REGION Network 36: LT-502 BUFF
   RUNG wire#powerrail
      Contact( "AlwaysTRUE" )
      wire#w1
      { S7_Templates := "SrcType := Real" } LT_Contact(in1 := "AI SCALING DB".PV."LEVEL TRANSMITTER 502", in2 := "AI SCALING DB"."LT-502 SET VALVE".LL)
      { S7_Templates := "time_type := Time" } "IEC_Timer_0_DB_30".TON(pt := T#3S, et =>)
      Move(in := 1, out1 => "AI SCALING DB"."LT-502".LOW_BUFF)
   END_RUNG
   RUNG wire#w1
      { S7_Templates := "SrcType := Real" } GE_Contact(in1 := "AI SCALING DB".PV."LEVEL TRANSMITTER 502", in2 := "AI SCALING DB"."LT-502 SET VALVE".L)
      { S7_Templates := "time_type := Time" } "IEC_Timer_0_DB_31".TON(pt := T#3S, et =>)
      Move(in := 2, out1 => "AI SCALING DB"."LT-502".LOW_BUFF)
   END_RUNG
   RUNG wire#w1
      { S7_Templates := "SrcType := Real" } LT_Contact(in1 := "AI SCALING DB".PV."LEVEL TRANSMITTER 502", in2 := "AI SCALING DB"."LT-502 SET VALVE".H)
      { S7_Templates := "time_type := Time" } "IEC_Timer_0_DB_32".TON(pt := T#3S, et =>)
      Move(in := 3, out1 => "AI SCALING DB"."LT-502".HIGH_BUFF)
   END_RUNG
   RUNG wire#w1
      { S7_Templates := "SrcType := Real" } GE_Contact(in1 := "AI SCALING DB".PV."LEVEL TRANSMITTER 502", in2 := "AI SCALING DB"."LT-502 SET VALVE".HH)
      { S7_Templates := "time_type := Time" } "IEC_Timer_0_DB_33".TON(pt := T#3S, et =>)
      Move(in := 4, out1 => "AI SCALING DB"."LT-502".HIGH_BUFF)
   END_RUNG
   // the same network as SCL:
   "IEC_Timer_0_DB_30".TON(IN := "AlwaysTRUE" AND ("AI SCALING DB".PV."LEVEL TRANSMITTER 502" < "AI SCALING DB"."LT-502 SET VALVE".LL),
                           PT := T#3S);
   IF "IEC_Timer_0_DB_30".Q THEN "AI SCALING DB"."LT-502".LOW_BUFF := 1; END_IF;
   "IEC_Timer_0_DB_31".TON(IN := "AlwaysTRUE" AND ("AI SCALING DB".PV."LEVEL TRANSMITTER 502" >= "AI SCALING DB"."LT-502 SET VALVE".L),
                           PT := T#3S);
   IF "IEC_Timer_0_DB_31".Q THEN "AI SCALING DB"."LT-502".LOW_BUFF := 2; END_IF;
   "IEC_Timer_0_DB_32".TON(IN := "AlwaysTRUE" AND ("AI SCALING DB".PV."LEVEL TRANSMITTER 502" < "AI SCALING DB"."LT-502 SET VALVE".H),
                           PT := T#3S);
   IF "IEC_Timer_0_DB_32".Q THEN "AI SCALING DB"."LT-502".HIGH_BUFF := 3; END_IF;
   "IEC_Timer_0_DB_33".TON(IN := "AlwaysTRUE" AND ("AI SCALING DB".PV."LEVEL TRANSMITTER 502" >= "AI SCALING DB"."LT-502 SET VALVE".HH),
                           PT := T#3S);
   IF "IEC_Timer_0_DB_33".Q THEN "AI SCALING DB"."LT-502".HIGH_BUFF := 4; END_IF;
END_REGION

REGION Network 38: "DataToSlave".DATA1."LT-502 BUFFER"."LT-502 LOW"
   RUNG wire#powerrail
      Move(in := "AI SCALING DB"."LT-502".LOW_BUFF, out1 => "DataToMaster".DATA1."LT-502".LOW_BUFF)
   END_RUNG
   // the same network as SCL:
   "DataToMaster".DATA1."LT-502".LOW_BUFF := "AI SCALING DB"."LT-502".LOW_BUFF;
END_REGION

REGION Network 39: "DataToSlave".DATA1."LT-502 BUFFER"."LT-502 HIGH
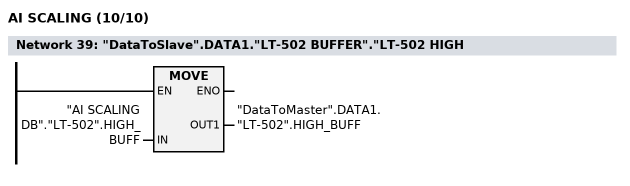
   RUNG wire#powerrail
      Move(in := "AI SCALING DB"."LT-502".HIGH_BUFF, out1 => "DataToMaster".DATA1."LT-502".HIGH_BUFF)
   END_RUNG
   // the same network as SCL:
   "DataToMaster".DATA1."LT-502".HIGH_BUFF := "AI SCALING DB"."LT-502".HIGH_BUFF;
END_REGION
END_FUNCTION

FUNCTION_BLOCK "SCALE"   // FB1, LAD
{ S7_Optimized_Access := 'TRUE' }
// stored: MemoryReserve 100, SetENOAutomatically false
   VAR_INPUT
      "SCALE MIN" : Real;
      "SCALE MAX" : Real;
      INPUT : Int;
      "RAW MIN" : Int;
      "RAW MAX" : Int;
   END_VAR
   VAR_OUTPUT
      "PV VALUE" : Real;
   END_VAR
   VAR_TEMP
      NORMX : Real;
   END_VAR
BEGIN

REGION Network 1
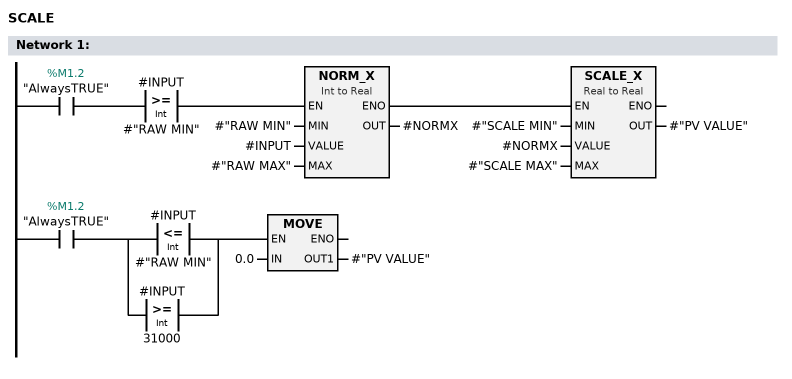
   RUNG wire#powerrail
      Contact( "AlwaysTRUE" )
      { S7_Templates := "SrcType := Int" } GE_Contact(in1 := #INPUT, in2 := #"RAW MIN")
      { S7_Templates := "[SrcType := Int, DestType := Real]" } Normalize(min := #"RAW MIN", value := #INPUT, max := #"RAW MAX", out => #NORMX)
      { S7_Templates := "[SrcType := Real, DestType := Real]" } Scale(min := #"SCALE MIN", value := #NORMX, max := #"SCALE MAX", out => #"PV VALUE")
   END_RUNG
   RUNG wire#powerrail
      Contact( "AlwaysTRUE" )
      wire#w1
      { S7_Templates := "SrcType := Int" } LE_Contact(in1 := #INPUT, in2 := #"RAW MIN")
      wire#w2
      Move(in := 0.0, out1 => #"PV VALUE")
   END_RUNG
   RUNG wire#w1
      { S7_Templates := "SrcType := Int" } GE_Contact(in1 := #INPUT, in2 := 31000)
   END_RUNG wire#w2
   // the same network as SCL:
   IF "AlwaysTRUE" AND (#INPUT >= #"RAW MIN") THEN
       #NORMX := NORM_X(MIN := #"RAW MIN", VALUE := #INPUT, MAX := #"RAW MAX");
       #"PV VALUE" := SCALE_X(MIN := #"SCALE MIN", VALUE := #NORMX, MAX := #"SCALE MAX");
   END_IF;
   IF "AlwaysTRUE" AND ((#INPUT <= #"RAW MIN") OR (#INPUT >= 31000)) THEN #"PV VALUE" := 0.0; END_IF;
END_REGION
END_FUNCTION_BLOCK

FUNCTION "INPUT MAPING" : Void   // FC1, LAD
{ S7_Optimized_Access := 'TRUE' }
// stored: SetENOAutomatically false
BEGIN

REGION Network 1: "CPU RUN"
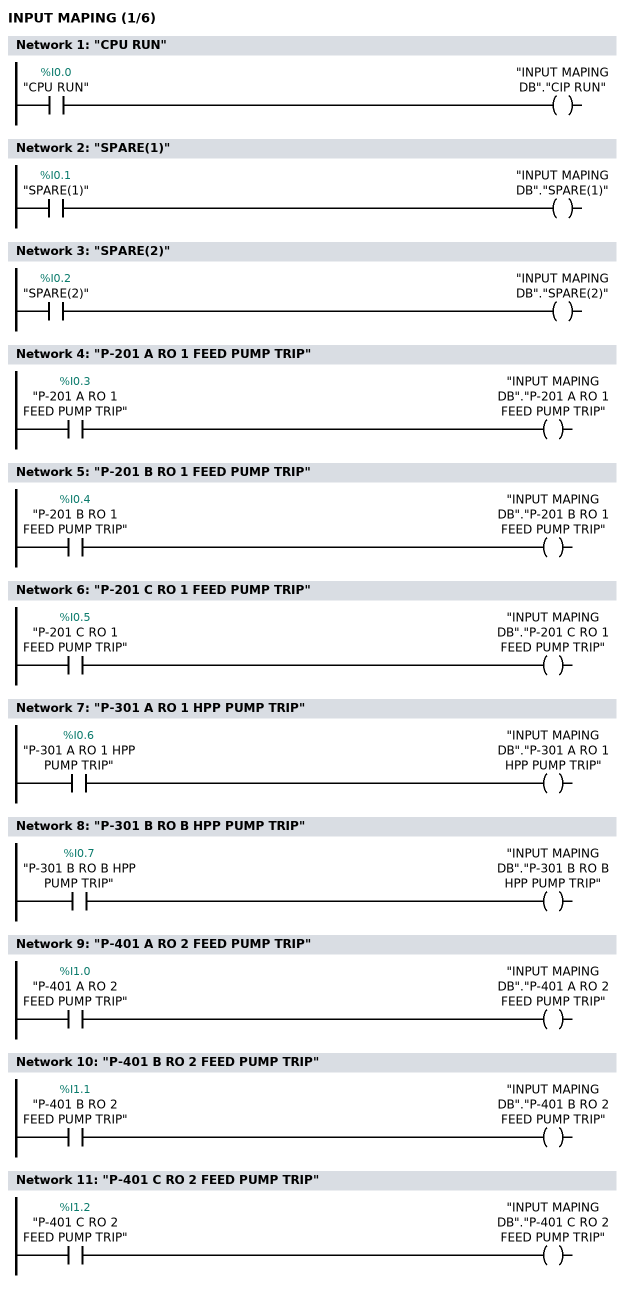
   RUNG wire#powerrail
      Contact( "CPU RUN" )
      Coil( "INPUT MAPING DB"."CIP RUN" )
   END_RUNG
   // the same network as SCL:
   "INPUT MAPING DB"."CIP RUN" := "CPU RUN";
END_REGION

REGION Network 2: "SPARE(1)"
   RUNG wire#powerrail
      Contact( "SPARE(1)" )
      Coil( "INPUT MAPING DB"."SPARE(1)" )
   END_RUNG
   // the same network as SCL:
   "INPUT MAPING DB"."SPARE(1)" := "SPARE(1)";
END_REGION

REGION Network 3: "SPARE(2)"
   RUNG wire#powerrail
      Contact( "SPARE(2)" )
      Coil( "INPUT MAPING DB"."SPARE(2)" )
   END_RUNG
   // the same network as SCL:
   "INPUT MAPING DB"."SPARE(2)" := "SPARE(2)";
END_REGION

REGION Network 4: "P-201 A RO 1 FEED PUMP TRIP"
   RUNG wire#powerrail
      Contact( "P-201 A RO 1 FEED PUMP TRIP" )
      Coil( "INPUT MAPING DB"."P-201 A RO 1 FEED PUMP TRIP" )
   END_RUNG
   // the same network as SCL:
   "INPUT MAPING DB"."P-201 A RO 1 FEED PUMP TRIP" := "P-201 A RO 1 FEED PUMP TRIP";
END_REGION

REGION Network 5: "P-201 B RO 1 FEED PUMP TRIP"
   RUNG wire#powerrail
      Contact( "P-201 B RO 1 FEED PUMP TRIP" )
      Coil( "INPUT MAPING DB"."P-201 B RO 1 FEED PUMP TRIP" )
   END_RUNG
   // the same network as SCL:
   "INPUT MAPING DB"."P-201 B RO 1 FEED PUMP TRIP" := "P-201 B RO 1 FEED PUMP TRIP";
END_REGION

REGION Network 6: "P-201 C RO 1 FEED PUMP TRIP"
   RUNG wire#powerrail
      Contact( "P-201 C RO 1 FEED PUMP TRIP" )
      Coil( "INPUT MAPING DB"."P-201 C RO 1 FEED PUMP TRIP" )
   END_RUNG
   // the same network as SCL:
   "INPUT MAPING DB"."P-201 C RO 1 FEED PUMP TRIP" := "P-201 C RO 1 FEED PUMP TRIP";
END_REGION

REGION Network 7: "P-301 A RO 1 HPP PUMP TRIP"
   RUNG wire#powerrail
      Contact( "P-301 A RO 1 HPP PUMP TRIP" )
      Coil( "INPUT MAPING DB"."P-301 A RO 1 HPP PUMP TRIP" )
   END_RUNG
   // the same network as SCL:
   "INPUT MAPING DB"."P-301 A RO 1 HPP PUMP TRIP" := "P-301 A RO 1 HPP PUMP TRIP";
END_REGION

REGION Network 8: "P-301 B RO B HPP PUMP TRIP"
   RUNG wire#powerrail
      Contact( "P-301 B RO B HPP PUMP TRIP" )
      Coil( "INPUT MAPING DB"."P-301 B RO B HPP PUMP TRIP" )
   END_RUNG
   // the same network as SCL:
   "INPUT MAPING DB"."P-301 B RO B HPP PUMP TRIP" := "P-301 B RO B HPP PUMP TRIP";
END_REGION

REGION Network 9: "P-401 A RO 2 FEED PUMP TRIP"
   RUNG wire#powerrail
      Contact( "P-401 A RO 2 FEED PUMP TRIP" )
      Coil( "INPUT MAPING DB"."P-401 A RO 2 FEED PUMP TRIP" )
   END_RUNG
   // the same network as SCL:
   "INPUT MAPING DB"."P-401 A RO 2 FEED PUMP TRIP" := "P-401 A RO 2 FEED PUMP TRIP";
END_REGION

REGION Network 10: "P-401 B RO 2 FEED PUMP TRIP"
   RUNG wire#powerrail
      Contact( "P-401 B RO 2 FEED PUMP TRIP" )
      Coil( "INPUT MAPING DB"."P-401 B RO 2 FEED PUMP TRIP" )
   END_RUNG
   // the same network as SCL:
   "INPUT MAPING DB"."P-401 B RO 2 FEED PUMP TRIP" := "P-401 B RO 2 FEED PUMP TRIP";
END_REGION

REGION Network 11: "P-401 C RO 2 FEED PUMP TRIP"
   RUNG wire#powerrail
      Contact( "P-401 C RO 2 FEED PUMP TRIP" )
      Coil( "INPUT MAPING DB"."P-401 C RO 2 FEED PUMP TRIP" )
   END_RUNG
   // the same network as SCL:
   "INPUT MAPING DB"."P-401 C RO 2 FEED PUMP TRIP" := "P-401 C RO 2 FEED PUMP TRIP";
END_REGION

REGION Network 12: "P 401 A RO 2 HPP PUMP TRIP"
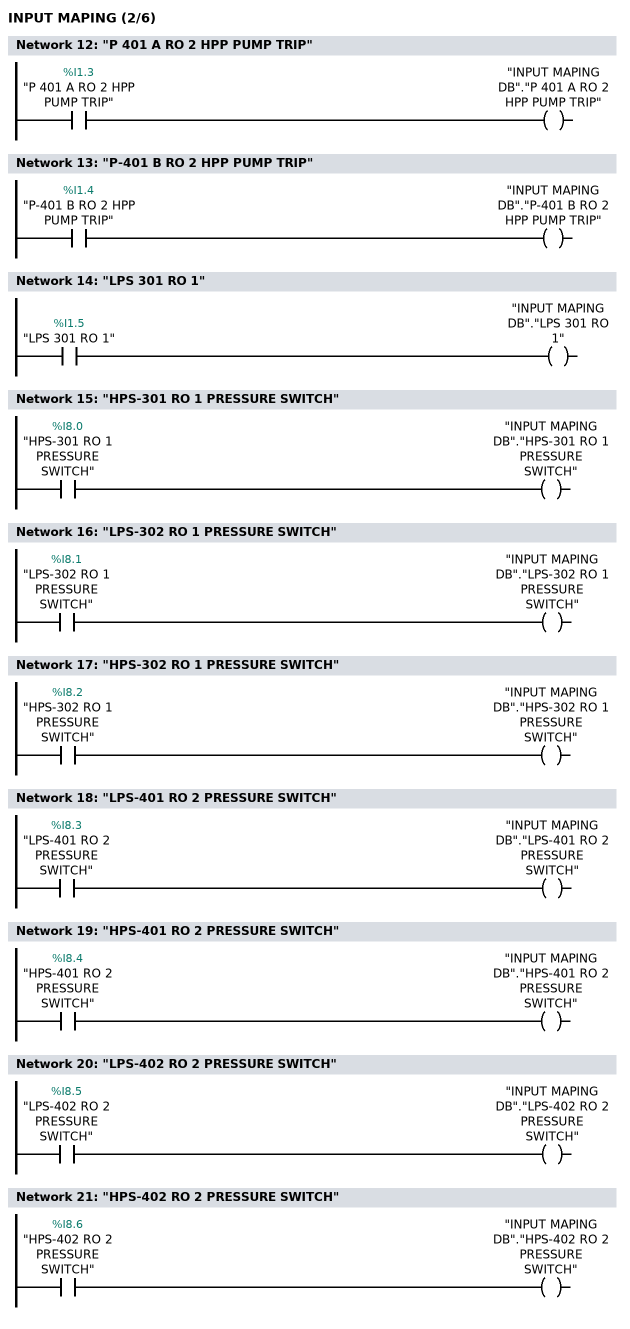
   RUNG wire#powerrail
      Contact( "P 401 A RO 2 HPP PUMP TRIP" )
      Coil( "INPUT MAPING DB"."P 401 A RO 2 HPP PUMP TRIP" )
   END_RUNG
   // the same network as SCL:
   "INPUT MAPING DB"."P 401 A RO 2 HPP PUMP TRIP" := "P 401 A RO 2 HPP PUMP TRIP";
END_REGION

REGION Network 13: "P-401 B RO 2 HPP PUMP TRIP"
   RUNG wire#powerrail
      Contact( "P-401 B RO 2 HPP PUMP TRIP" )
      Coil( "INPUT MAPING DB"."P-401 B RO 2 HPP PUMP TRIP" )
   END_RUNG
   // the same network as SCL:
   "INPUT MAPING DB"."P-401 B RO 2 HPP PUMP TRIP" := "P-401 B RO 2 HPP PUMP TRIP";
END_REGION

REGION Network 14: "LPS 301 RO 1"
   RUNG wire#powerrail
      Contact( "LPS 301 RO 1" )
      Coil( "INPUT MAPING DB"."LPS 301 RO 1" )
   END_RUNG
   // the same network as SCL:
   "INPUT MAPING DB"."LPS 301 RO 1" := "LPS 301 RO 1";
END_REGION

REGION Network 15: "HPS-301 RO 1 PRESSURE SWITCH"
   RUNG wire#powerrail
      Contact( "HPS-301 RO 1 PRESSURE SWITCH" )
      Coil( "INPUT MAPING DB"."HPS-301 RO 1 PRESSURE SWITCH" )
   END_RUNG
   // the same network as SCL:
   "INPUT MAPING DB"."HPS-301 RO 1 PRESSURE SWITCH" := "HPS-301 RO 1 PRESSURE SWITCH";
END_REGION

REGION Network 16: "LPS-302 RO 1 PRESSURE SWITCH"
   RUNG wire#powerrail
      Contact( "LPS-302 RO 1 PRESSURE SWITCH" )
      Coil( "INPUT MAPING DB"."LPS-302 RO 1 PRESSURE SWITCH" )
   END_RUNG
   // the same network as SCL:
   "INPUT MAPING DB"."LPS-302 RO 1 PRESSURE SWITCH" := "LPS-302 RO 1 PRESSURE SWITCH";
END_REGION

REGION Network 17: "HPS-302 RO 1 PRESSURE SWITCH"
   RUNG wire#powerrail
      Contact( "HPS-302 RO 1 PRESSURE SWITCH" )
      Coil( "INPUT MAPING DB"."HPS-302 RO 1 PRESSURE SWITCH" )
   END_RUNG
   // the same network as SCL:
   "INPUT MAPING DB"."HPS-302 RO 1 PRESSURE SWITCH" := "HPS-302 RO 1 PRESSURE SWITCH";
END_REGION

REGION Network 18: "LPS-401 RO 2 PRESSURE SWITCH"
   RUNG wire#powerrail
      Contact( "LPS-401 RO 2 PRESSURE SWITCH" )
      Coil( "INPUT MAPING DB"."LPS-401 RO 2 PRESSURE SWITCH" )
   END_RUNG
   // the same network as SCL:
   "INPUT MAPING DB"."LPS-401 RO 2 PRESSURE SWITCH" := "LPS-401 RO 2 PRESSURE SWITCH";
END_REGION

REGION Network 19: "HPS-401 RO 2 PRESSURE SWITCH"
   RUNG wire#powerrail
      Contact( "HPS-401 RO 2 PRESSURE SWITCH" )
      Coil( "INPUT MAPING DB"."HPS-401 RO 2 PRESSURE SWITCH" )
   END_RUNG
   // the same network as SCL:
   "INPUT MAPING DB"."HPS-401 RO 2 PRESSURE SWITCH" := "HPS-401 RO 2 PRESSURE SWITCH";
END_REGION

REGION Network 20: "LPS-402 RO 2 PRESSURE SWITCH"
   RUNG wire#powerrail
      Contact( "LPS-402 RO 2 PRESSURE SWITCH" )
      Coil( "INPUT MAPING DB"."LPS-402 RO 2 PRESSURE SWITCH" )
   END_RUNG
   // the same network as SCL:
   "INPUT MAPING DB"."LPS-402 RO 2 PRESSURE SWITCH" := "LPS-402 RO 2 PRESSURE SWITCH";
END_REGION

REGION Network 21: "HPS-402 RO 2 PRESSURE SWITCH"
   RUNG wire#powerrail
      Contact( "HPS-402 RO 2 PRESSURE SWITCH" )
      Coil( "INPUT MAPING DB"."HPS-402 RO 2 PRESSURE SWITCH" )
   END_RUNG
   // the same network as SCL:
   "INPUT MAPING DB"."HPS-402 RO 2 PRESSURE SWITCH" := "HPS-402 RO 2 PRESSURE SWITCH";
END_REGION

REGION Network 22: "DP-703 RO 1 DOSER LEVEL SWITCH"
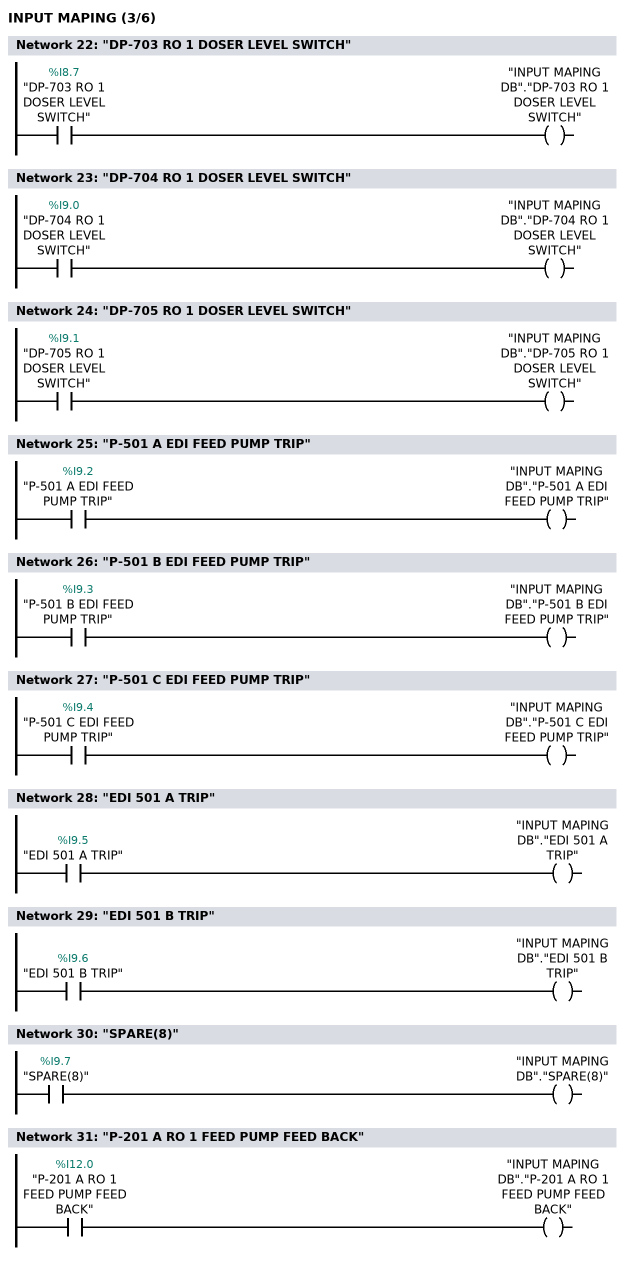
   RUNG wire#powerrail
      Contact( "DP-703 RO 1 DOSER LEVEL SWITCH" )
      Coil( "INPUT MAPING DB"."DP-703 RO 1 DOSER LEVEL SWITCH" )
   END_RUNG
   // the same network as SCL:
   "INPUT MAPING DB"."DP-703 RO 1 DOSER LEVEL SWITCH" := "DP-703 RO 1 DOSER LEVEL SWITCH";
END_REGION

REGION Network 23: "DP-704 RO 1 DOSER LEVEL SWITCH"
   RUNG wire#powerrail
      Contact( "DP-704 RO 1 DOSER LEVEL SWITCH" )
      Coil( "INPUT MAPING DB"."DP-704 RO 1 DOSER LEVEL SWITCH" )
   END_RUNG
   // the same network as SCL:
   "INPUT MAPING DB"."DP-704 RO 1 DOSER LEVEL SWITCH" := "DP-704 RO 1 DOSER LEVEL SWITCH";
END_REGION

REGION Network 24: "DP-705 RO 1 DOSER LEVEL SWITCH"
   RUNG wire#powerrail
      Contact( "DP-705 RO 1 DOSER LEVEL SWITCH" )
      Coil( "INPUT MAPING DB"."DP-705 RO 1 DOSER LEVEL SWITCH" )
   END_RUNG
   // the same network as SCL:
   "INPUT MAPING DB"."DP-705 RO 1 DOSER LEVEL SWITCH" := "DP-705 RO 1 DOSER LEVEL SWITCH";
END_REGION

REGION Network 25: "P-501 A EDI FEED PUMP TRIP"
   RUNG wire#powerrail
      Contact( "P-501 A EDI FEED PUMP TRIP" )
      Coil( "INPUT MAPING DB"."P-501 A EDI FEED PUMP TRIP" )
   END_RUNG
   // the same network as SCL:
   "INPUT MAPING DB"."P-501 A EDI FEED PUMP TRIP" := "P-501 A EDI FEED PUMP TRIP";
END_REGION

REGION Network 26: "P-501 B EDI FEED PUMP TRIP"
   RUNG wire#powerrail
      Contact( "P-501 B EDI FEED PUMP TRIP" )
      Coil( "INPUT MAPING DB"."P-501 B EDI FEED PUMP TRIP" )
   END_RUNG
   // the same network as SCL:
   "INPUT MAPING DB"."P-501 B EDI FEED PUMP TRIP" := "P-501 B EDI FEED PUMP TRIP";
END_REGION

REGION Network 27: "P-501 C EDI FEED PUMP TRIP"
   RUNG wire#powerrail
      Contact( "P-501 C EDI FEED PUMP TRIP" )
      Coil( "INPUT MAPING DB"."P-501 C EDI FEED PUMP TRIP" )
   END_RUNG
   // the same network as SCL:
   "INPUT MAPING DB"."P-501 C EDI FEED PUMP TRIP" := "P-501 C EDI FEED PUMP TRIP";
END_REGION

REGION Network 28: "EDI 501 A TRIP"
   RUNG wire#powerrail
      Contact( "EDI 501 A TRIP" )
      Coil( "INPUT MAPING DB"."EDI 501 A TRIP" )
   END_RUNG
   // the same network as SCL:
   "INPUT MAPING DB"."EDI 501 A TRIP" := "EDI 501 A TRIP";
END_REGION

REGION Network 29: "EDI 501 B TRIP"
   RUNG wire#powerrail
      Contact( "EDI 501 B TRIP" )
      Coil( "INPUT MAPING DB"."EDI 501 B TRIP" )
   END_RUNG
   // the same network as SCL:
   "INPUT MAPING DB"."EDI 501 B TRIP" := "EDI 501 B TRIP";
END_REGION

REGION Network 30: "SPARE(8)"
   RUNG wire#powerrail
      Contact( "SPARE(8)" )
      Coil( "INPUT MAPING DB"."SPARE(8)" )
   END_RUNG
   // the same network as SCL:
   "INPUT MAPING DB"."SPARE(8)" := "SPARE(8)";
END_REGION

REGION Network 31: "P-201 A RO 1 FEED PUMP FEED BACK"
   RUNG wire#powerrail
      Contact( "P-201 A RO 1 FEED PUMP FEED BACK" )
      Coil( "INPUT MAPING DB"."P-201 A RO 1 FEED PUMP FEED BACK" )
   END_RUNG
   // the same network as SCL:
   "INPUT MAPING DB"."P-201 A RO 1 FEED PUMP FEED BACK" := "P-201 A RO 1 FEED PUMP FEED BACK";
END_REGION

REGION Network 32: "P-201 B RO 1 FEED PUMP FEED BACK"
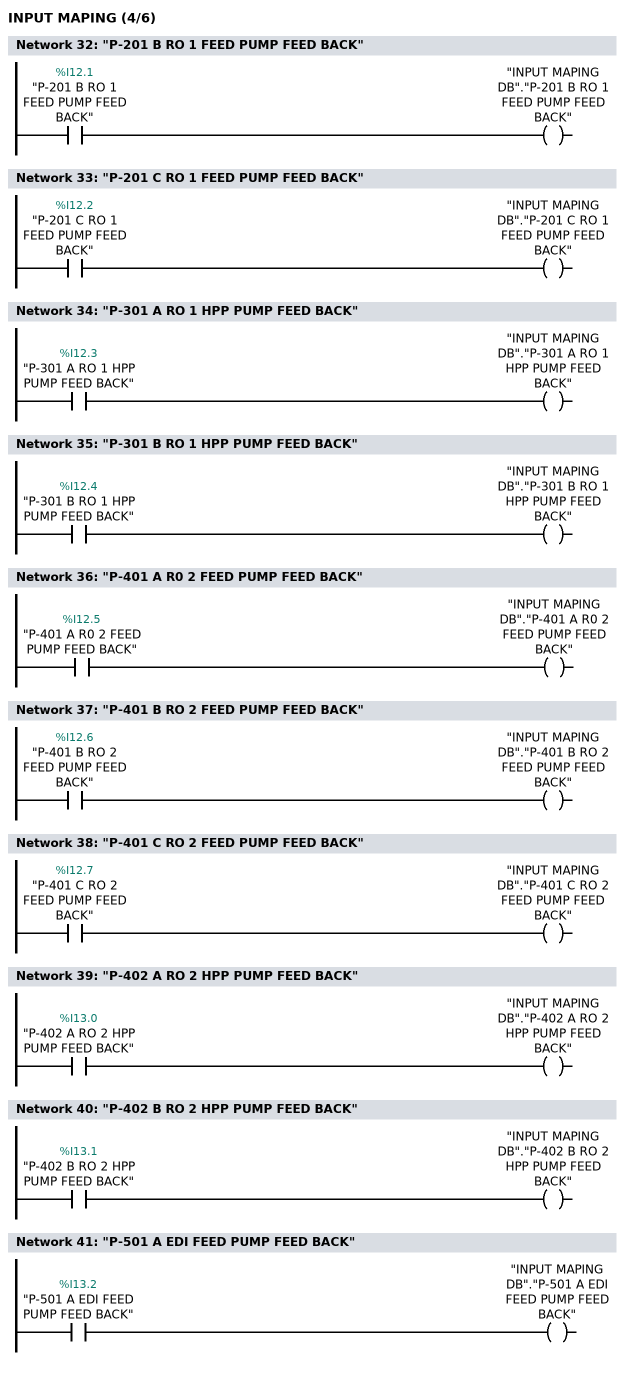
   RUNG wire#powerrail
      Contact( "P-201 B RO 1 FEED PUMP FEED BACK" )
      Coil( "INPUT MAPING DB"."P-201 B RO 1 FEED PUMP FEED BACK" )
   END_RUNG
   // the same network as SCL:
   "INPUT MAPING DB"."P-201 B RO 1 FEED PUMP FEED BACK" := "P-201 B RO 1 FEED PUMP FEED BACK";
END_REGION

REGION Network 33: "P-201 C RO 1 FEED PUMP FEED BACK"
   RUNG wire#powerrail
      Contact( "P-201 C RO 1 FEED PUMP FEED BACK" )
      Coil( "INPUT MAPING DB"."P-201 C RO 1 FEED PUMP FEED BACK" )
   END_RUNG
   // the same network as SCL:
   "INPUT MAPING DB"."P-201 C RO 1 FEED PUMP FEED BACK" := "P-201 C RO 1 FEED PUMP FEED BACK";
END_REGION

REGION Network 34: "P-301 A RO 1 HPP PUMP FEED BACK"
   RUNG wire#powerrail
      Contact( "P-301 A RO 1 HPP PUMP FEED BACK" )
      Coil( "INPUT MAPING DB"."P-301 A RO 1 HPP PUMP FEED BACK" )
   END_RUNG
   // the same network as SCL:
   "INPUT MAPING DB"."P-301 A RO 1 HPP PUMP FEED BACK" := "P-301 A RO 1 HPP PUMP FEED BACK";
END_REGION

REGION Network 35: "P-301 B RO 1 HPP PUMP FEED BACK"
   RUNG wire#powerrail
      Contact( "P-301 B RO 1 HPP PUMP FEED BACK" )
      Coil( "INPUT MAPING DB"."P-301 B RO 1 HPP PUMP FEED BACK" )
   END_RUNG
   // the same network as SCL:
   "INPUT MAPING DB"."P-301 B RO 1 HPP PUMP FEED BACK" := "P-301 B RO 1 HPP PUMP FEED BACK";
END_REGION

REGION Network 36: "P-401 A R0 2 FEED PUMP FEED BACK"
   RUNG wire#powerrail
      Contact( "P-401 A R0 2 FEED PUMP FEED BACK" )
      Coil( "INPUT MAPING DB"."P-401 A R0 2 FEED PUMP FEED BACK" )
   END_RUNG
   // the same network as SCL:
   "INPUT MAPING DB"."P-401 A R0 2 FEED PUMP FEED BACK" := "P-401 A R0 2 FEED PUMP FEED BACK";
END_REGION

REGION Network 37: "P-401 B RO 2 FEED PUMP FEED BACK"
   RUNG wire#powerrail
      Contact( "P-401 B RO 2 FEED PUMP FEED BACK" )
      Coil( "INPUT MAPING DB"."P-401 B RO 2 FEED PUMP FEED BACK" )
   END_RUNG
   // the same network as SCL:
   "INPUT MAPING DB"."P-401 B RO 2 FEED PUMP FEED BACK" := "P-401 B RO 2 FEED PUMP FEED BACK";
END_REGION

REGION Network 38: "P-401 C RO 2 FEED PUMP FEED BACK"
   RUNG wire#powerrail
      Contact( "P-401 C RO 2 FEED PUMP FEED BACK" )
      Coil( "INPUT MAPING DB"."P-401 C RO 2 FEED PUMP FEED BACK" )
   END_RUNG
   // the same network as SCL:
   "INPUT MAPING DB"."P-401 C RO 2 FEED PUMP FEED BACK" := "P-401 C RO 2 FEED PUMP FEED BACK";
END_REGION

REGION Network 39: "P-402 A RO 2 HPP PUMP FEED BACK"
   RUNG wire#powerrail
      Contact( "P-402 A RO 2 HPP PUMP FEED BACK" )
      Coil( "INPUT MAPING DB"."P-402 A RO 2 HPP PUMP FEED BACK" )
   END_RUNG
   // the same network as SCL:
   "INPUT MAPING DB"."P-402 A RO 2 HPP PUMP FEED BACK" := "P-402 A RO 2 HPP PUMP FEED BACK";
END_REGION

REGION Network 40: "P-402 B RO 2 HPP PUMP FEED BACK"
   RUNG wire#powerrail
      Contact( "P-402 B RO 2 HPP PUMP FEED BACK" )
      Coil( "INPUT MAPING DB"."P-402 B RO 2 HPP PUMP FEED BACK" )
   END_RUNG
   // the same network as SCL:
   "INPUT MAPING DB"."P-402 B RO 2 HPP PUMP FEED BACK" := "P-402 B RO 2 HPP PUMP FEED BACK";
END_REGION

REGION Network 41: "P-501 A EDI FEED PUMP FEED BACK"
   RUNG wire#powerrail
      Contact( "P-501 A EDI FEED PUMP FEED BACK" )
      Coil( "INPUT MAPING DB"."P-501 A EDI FEED PUMP FEED BACK" )
   END_RUNG
   // the same network as SCL:
   "INPUT MAPING DB"."P-501 A EDI FEED PUMP FEED BACK" := "P-501 A EDI FEED PUMP FEED BACK";
END_REGION

REGION Network 42: "P-501 B EDI FEED PUMP FEED BACK"
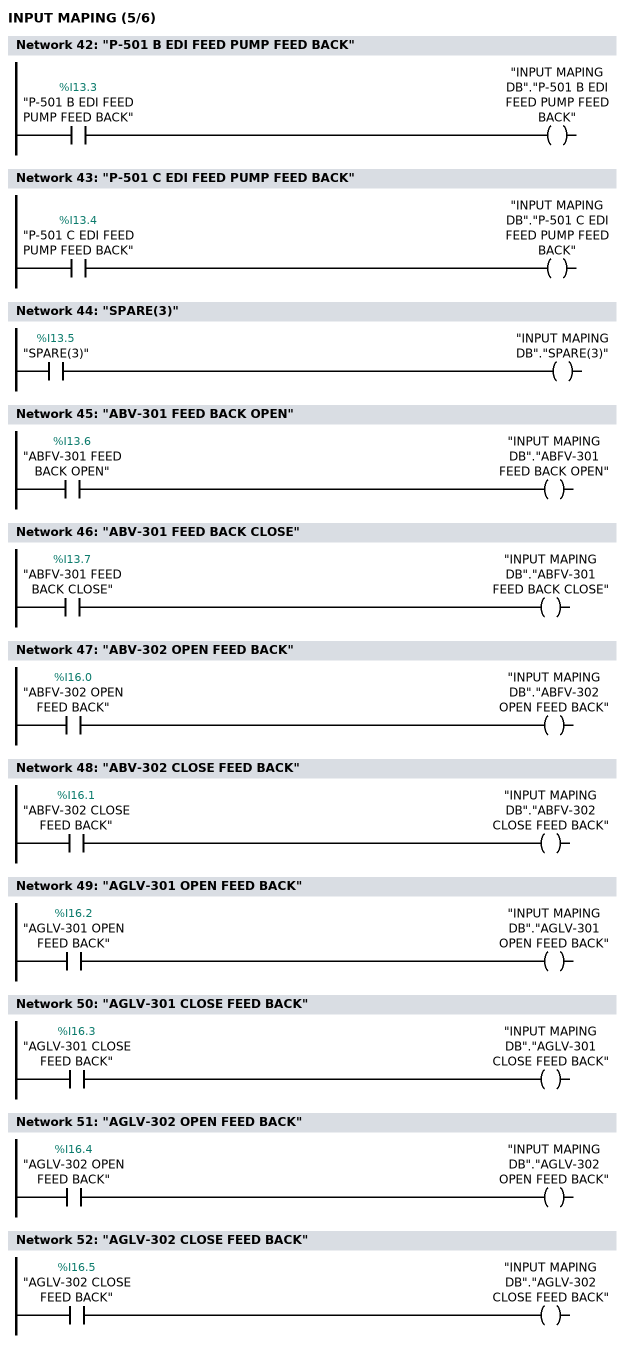
   RUNG wire#powerrail
      Contact( "P-501 B EDI FEED PUMP FEED BACK" )
      Coil( "INPUT MAPING DB"."P-501 B EDI FEED PUMP FEED BACK" )
   END_RUNG
   // the same network as SCL:
   "INPUT MAPING DB"."P-501 B EDI FEED PUMP FEED BACK" := "P-501 B EDI FEED PUMP FEED BACK";
END_REGION

REGION Network 43: "P-501 C EDI FEED PUMP FEED BACK"
   RUNG wire#powerrail
      Contact( "P-501 C EDI FEED PUMP FEED BACK" )
      Coil( "INPUT MAPING DB"."P-501 C EDI FEED PUMP FEED BACK" )
   END_RUNG
   // the same network as SCL:
   "INPUT MAPING DB"."P-501 C EDI FEED PUMP FEED BACK" := "P-501 C EDI FEED PUMP FEED BACK";
END_REGION

REGION Network 44: "SPARE(3)"
   RUNG wire#powerrail
      Contact( "SPARE(3)" )
      Coil( "INPUT MAPING DB"."SPARE(3)" )
   END_RUNG
   // the same network as SCL:
   "INPUT MAPING DB"."SPARE(3)" := "SPARE(3)";
END_REGION

REGION Network 45: "ABV-301 FEED BACK OPEN"
   RUNG wire#powerrail
      Contact( "ABFV-301 FEED BACK OPEN" )
      Coil( "INPUT MAPING DB"."ABFV-301 FEED BACK OPEN" )
   END_RUNG
   // the same network as SCL:
   "INPUT MAPING DB"."ABFV-301 FEED BACK OPEN" := "ABFV-301 FEED BACK OPEN";
END_REGION

REGION Network 46: "ABV-301 FEED BACK CLOSE"
   RUNG wire#powerrail
      Contact( "ABFV-301 FEED BACK CLOSE" )
      Coil( "INPUT MAPING DB"."ABFV-301 FEED BACK CLOSE" )
   END_RUNG
   // the same network as SCL:
   "INPUT MAPING DB"."ABFV-301 FEED BACK CLOSE" := "ABFV-301 FEED BACK CLOSE";
END_REGION

REGION Network 47: "ABV-302 OPEN FEED BACK"
   RUNG wire#powerrail
      Contact( "ABFV-302 OPEN FEED BACK" )
      Coil( "INPUT MAPING DB"."ABFV-302 OPEN FEED BACK" )
   END_RUNG
   // the same network as SCL:
   "INPUT MAPING DB"."ABFV-302 OPEN FEED BACK" := "ABFV-302 OPEN FEED BACK";
END_REGION

REGION Network 48: "ABV-302 CLOSE FEED BACK"
   RUNG wire#powerrail
      Contact( "ABFV-302 CLOSE FEED BACK" )
      Coil( "INPUT MAPING DB"."ABFV-302 CLOSE FEED BACK" )
   END_RUNG
   // the same network as SCL:
   "INPUT MAPING DB"."ABFV-302 CLOSE FEED BACK" := "ABFV-302 CLOSE FEED BACK";
END_REGION

REGION Network 49: "AGLV-301 OPEN FEED BACK"
   RUNG wire#powerrail
      Contact( "AGLV-301 OPEN FEED BACK" )
      Coil( "INPUT MAPING DB"."AGLV-301 OPEN FEED BACK" )
   END_RUNG
   // the same network as SCL:
   "INPUT MAPING DB"."AGLV-301 OPEN FEED BACK" := "AGLV-301 OPEN FEED BACK";
END_REGION

REGION Network 50: "AGLV-301 CLOSE FEED BACK"
   RUNG wire#powerrail
      Contact( "AGLV-301 CLOSE FEED BACK" )
      Coil( "INPUT MAPING DB"."AGLV-301 CLOSE FEED BACK" )
   END_RUNG
   // the same network as SCL:
   "INPUT MAPING DB"."AGLV-301 CLOSE FEED BACK" := "AGLV-301 CLOSE FEED BACK";
END_REGION

REGION Network 51: "AGLV-302 OPEN FEED BACK"
   RUNG wire#powerrail
      Contact( "AGLV-302 OPEN FEED BACK" )
      Coil( "INPUT MAPING DB"."AGLV-302 OPEN FEED BACK" )
   END_RUNG
   // the same network as SCL:
   "INPUT MAPING DB"."AGLV-302 OPEN FEED BACK" := "AGLV-302 OPEN FEED BACK";
END_REGION

REGION Network 52: "AGLV-302 CLOSE FEED BACK"
   RUNG wire#powerrail
      Contact( "AGLV-302 CLOSE FEED BACK" )
      Coil( "INPUT MAPING DB"."AGLV-302 CLOSE FEED BACK" )
   END_RUNG
   // the same network as SCL:
   "INPUT MAPING DB"."AGLV-302 CLOSE FEED BACK" := "AGLV-302 CLOSE FEED BACK";
END_REGION

REGION Network 53: "AGLV-401 OPEN FEED BACK"
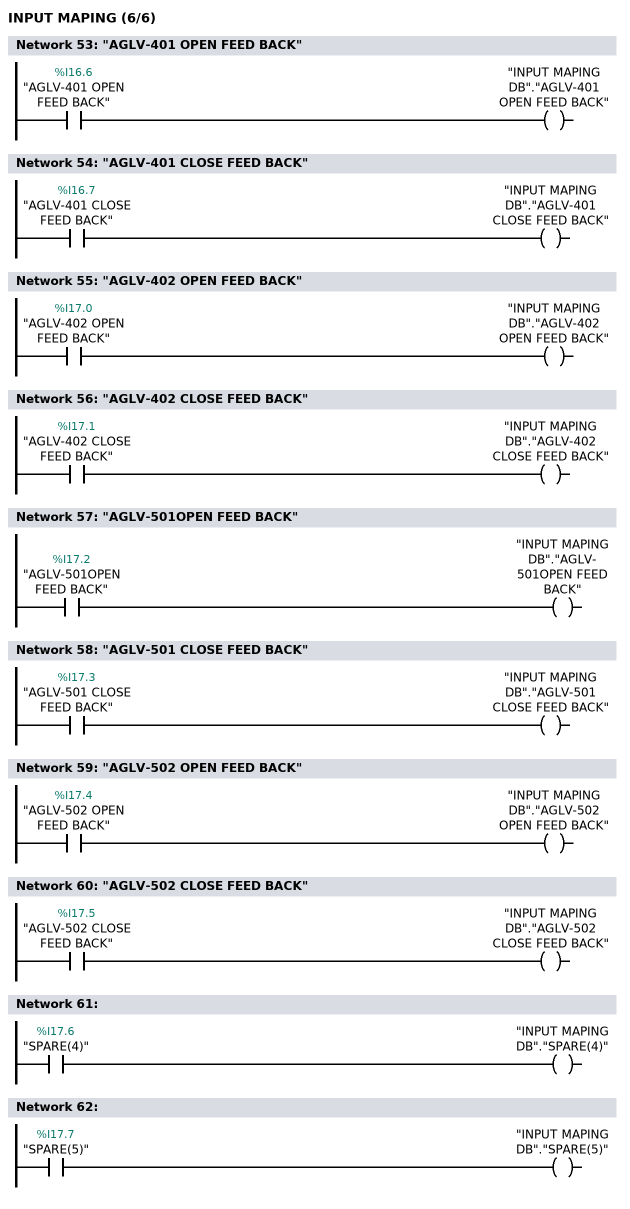
   RUNG wire#powerrail
      Contact( "AGLV-401 OPEN FEED BACK" )
      Coil( "INPUT MAPING DB"."AGLV-401 OPEN FEED BACK" )
   END_RUNG
   // the same network as SCL:
   "INPUT MAPING DB"."AGLV-401 OPEN FEED BACK" := "AGLV-401 OPEN FEED BACK";
END_REGION

REGION Network 54: "AGLV-401 CLOSE FEED BACK"
   RUNG wire#powerrail
      Contact( "AGLV-401 CLOSE FEED BACK" )
      Coil( "INPUT MAPING DB"."AGLV-401 CLOSE FEED BACK" )
   END_RUNG
   // the same network as SCL:
   "INPUT MAPING DB"."AGLV-401 CLOSE FEED BACK" := "AGLV-401 CLOSE FEED BACK";
END_REGION

REGION Network 55: "AGLV-402 OPEN FEED BACK"
   RUNG wire#powerrail
      Contact( "AGLV-402 OPEN FEED BACK" )
      Coil( "INPUT MAPING DB"."AGLV-402 OPEN FEED BACK" )
   END_RUNG
   // the same network as SCL:
   "INPUT MAPING DB"."AGLV-402 OPEN FEED BACK" := "AGLV-402 OPEN FEED BACK";
END_REGION

REGION Network 56: "AGLV-402 CLOSE FEED BACK"
   RUNG wire#powerrail
      Contact( "AGLV-402 CLOSE FEED BACK" )
      Coil( "INPUT MAPING DB"."AGLV-402 CLOSE FEED BACK" )
   END_RUNG
   // the same network as SCL:
   "INPUT MAPING DB"."AGLV-402 CLOSE FEED BACK" := "AGLV-402 CLOSE FEED BACK";
END_REGION

REGION Network 57: "AGLV-501OPEN FEED BACK"
   RUNG wire#powerrail
      Contact( "AGLV-501OPEN FEED BACK" )
      Coil( "INPUT MAPING DB"."AGLV-501OPEN FEED BACK" )
   END_RUNG
   // the same network as SCL:
   "INPUT MAPING DB"."AGLV-501OPEN FEED BACK" := "AGLV-501OPEN FEED BACK";
END_REGION

REGION Network 58: "AGLV-501 CLOSE FEED BACK"
   RUNG wire#powerrail
      Contact( "AGLV-501 CLOSE FEED BACK" )
      Coil( "INPUT MAPING DB"."AGLV-501 CLOSE FEED BACK" )
   END_RUNG
   // the same network as SCL:
   "INPUT MAPING DB"."AGLV-501 CLOSE FEED BACK" := "AGLV-501 CLOSE FEED BACK";
END_REGION

REGION Network 59: "AGLV-502 OPEN FEED BACK"
   RUNG wire#powerrail
      Contact( "AGLV-502 OPEN FEED BACK" )
      Coil( "INPUT MAPING DB"."AGLV-502 OPEN FEED BACK" )
   END_RUNG
   // the same network as SCL:
   "INPUT MAPING DB"."AGLV-502 OPEN FEED BACK" := "AGLV-502 OPEN FEED BACK";
END_REGION

REGION Network 60: "AGLV-502 CLOSE FEED BACK"
   RUNG wire#powerrail
      Contact( "AGLV-502 CLOSE FEED BACK" )
      Coil( "INPUT MAPING DB"."AGLV-502 CLOSE FEED BACK" )
   END_RUNG
   // the same network as SCL:
   "INPUT MAPING DB"."AGLV-502 CLOSE FEED BACK" := "AGLV-502 CLOSE FEED BACK";
END_REGION

REGION Network 61
   RUNG wire#powerrail
      Contact( "SPARE(4)" )
      Coil( "INPUT MAPING DB"."SPARE(4)" )
   END_RUNG
   // the same network as SCL:
   "INPUT MAPING DB"."SPARE(4)" := "SPARE(4)";
END_REGION

REGION Network 62
   RUNG wire#powerrail
      Contact( "SPARE(5)" )
      Coil( "INPUT MAPING DB"."SPARE(5)" )
   END_RUNG
   // the same network as SCL:
   "INPUT MAPING DB"."SPARE(5)" := "SPARE(5)";
END_REGION
END_FUNCTION

FUNCTION "OUTPUT MAPING" : Void   // FC2, LAD
{ S7_Optimized_Access := 'TRUE' }
// stored: SetENOAutomatically false
BEGIN

REGION Network 1: "P-202 A RO 1 FEED PUMP"
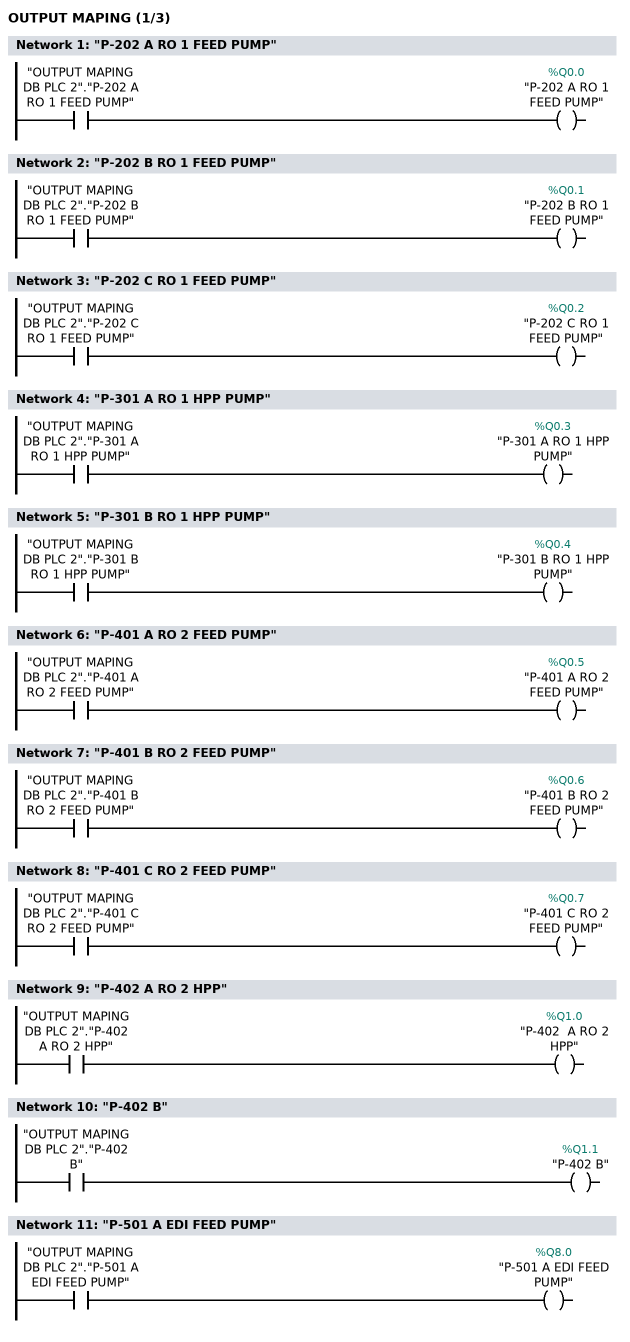
   RUNG wire#powerrail
      Contact( "OUTPUT MAPING DB PLC 2"."P-202 A RO 1 FEED PUMP" )
      Coil( "P-202 A RO 1 FEED PUMP" )
   END_RUNG
   // the same network as SCL:
   "P-202 A RO 1 FEED PUMP" := "OUTPUT MAPING DB PLC 2"."P-202 A RO 1 FEED PUMP";
END_REGION

REGION Network 2: "P-202 B RO 1 FEED PUMP"
   RUNG wire#powerrail
      Contact( "OUTPUT MAPING DB PLC 2"."P-202 B RO 1 FEED PUMP" )
      Coil( "P-202 B RO 1 FEED PUMP" )
   END_RUNG
   // the same network as SCL:
   "P-202 B RO 1 FEED PUMP" := "OUTPUT MAPING DB PLC 2"."P-202 B RO 1 FEED PUMP";
END_REGION

REGION Network 3: "P-202 C RO 1 FEED PUMP"
   RUNG wire#powerrail
      Contact( "OUTPUT MAPING DB PLC 2"."P-202 C RO 1 FEED PUMP" )
      Coil( "P-202 C RO 1 FEED PUMP" )
   END_RUNG
   // the same network as SCL:
   "P-202 C RO 1 FEED PUMP" := "OUTPUT MAPING DB PLC 2"."P-202 C RO 1 FEED PUMP";
END_REGION

REGION Network 4: "P-301 A RO 1 HPP PUMP"
   RUNG wire#powerrail
      Contact( "OUTPUT MAPING DB PLC 2"."P-301 A RO 1 HPP PUMP" )
      Coil( "P-301 A RO 1 HPP PUMP" )
   END_RUNG
   // the same network as SCL:
   "P-301 A RO 1 HPP PUMP" := "OUTPUT MAPING DB PLC 2"."P-301 A RO 1 HPP PUMP";
END_REGION

REGION Network 5: "P-301 B RO 1 HPP PUMP"
   RUNG wire#powerrail
      Contact( "OUTPUT MAPING DB PLC 2"."P-301 B RO 1 HPP PUMP" )
      Coil( "P-301 B RO 1 HPP PUMP" )
   END_RUNG
   // the same network as SCL:
   "P-301 B RO 1 HPP PUMP" := "OUTPUT MAPING DB PLC 2"."P-301 B RO 1 HPP PUMP";
END_REGION

REGION Network 6: "P-401 A RO 2 FEED PUMP"
   RUNG wire#powerrail
      Contact( "OUTPUT MAPING DB PLC 2"."P-401 A RO 2 FEED PUMP" )
      Coil( "P-401 A RO 2 FEED PUMP" )
   END_RUNG
   // the same network as SCL:
   "P-401 A RO 2 FEED PUMP" := "OUTPUT MAPING DB PLC 2"."P-401 A RO 2 FEED PUMP";
END_REGION

REGION Network 7: "P-401 B RO 2 FEED PUMP"
   RUNG wire#powerrail
      Contact( "OUTPUT MAPING DB PLC 2"."P-401 B RO 2 FEED PUMP" )
      Coil( "P-401 B RO 2 FEED PUMP" )
   END_RUNG
   // the same network as SCL:
   "P-401 B RO 2 FEED PUMP" := "OUTPUT MAPING DB PLC 2"."P-401 B RO 2 FEED PUMP";
END_REGION

REGION Network 8: "P-401 C RO 2 FEED PUMP"
   RUNG wire#powerrail
      Contact( "OUTPUT MAPING DB PLC 2"."P-401 C RO 2 FEED PUMP" )
      Coil( "P-401 C RO 2 FEED PUMP" )
   END_RUNG
   // the same network as SCL:
   "P-401 C RO 2 FEED PUMP" := "OUTPUT MAPING DB PLC 2"."P-401 C RO 2 FEED PUMP";
END_REGION

REGION Network 9: "P-402 A RO 2 HPP"
   RUNG wire#powerrail
      Contact( "OUTPUT MAPING DB PLC 2"."P-402  A RO 2 HPP" )
      Coil( "P-402  A RO 2 HPP" )
   END_RUNG
   // the same network as SCL:
   "P-402  A RO 2 HPP" := "OUTPUT MAPING DB PLC 2"."P-402  A RO 2 HPP";
END_REGION

REGION Network 10: "P-402 B"
   RUNG wire#powerrail
      Contact( "OUTPUT MAPING DB PLC 2"."P-402 B" )
      Coil( "P-402 B" )
   END_RUNG
   // the same network as SCL:
   "P-402 B" := "OUTPUT MAPING DB PLC 2"."P-402 B";
END_REGION

REGION Network 11: "P-501 A EDI FEED PUMP"
   RUNG wire#powerrail
      Contact( "OUTPUT MAPING DB PLC 2"."P-501 A EDI FEED PUMP" )
      Coil( "P-501 A EDI FEED PUMP" )
   END_RUNG
   // the same network as SCL:
   "P-501 A EDI FEED PUMP" := "OUTPUT MAPING DB PLC 2"."P-501 A EDI FEED PUMP";
END_REGION

REGION Network 12: "P-501 B EDI FEED PUMP"
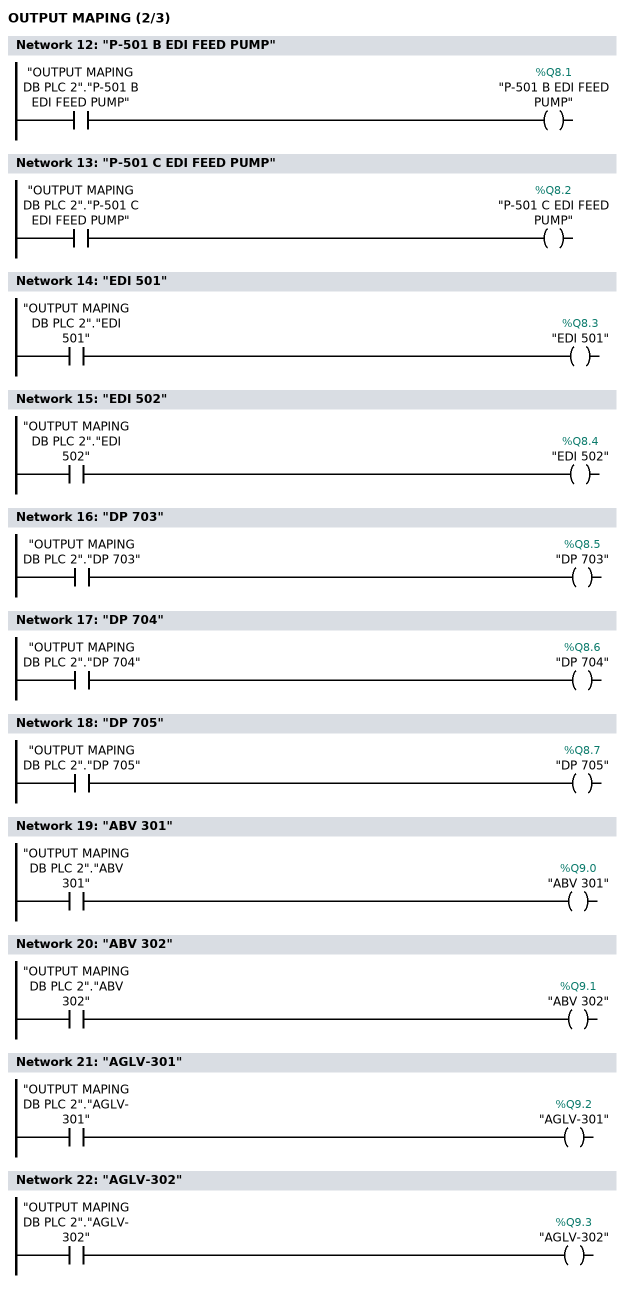
   RUNG wire#powerrail
      Contact( "OUTPUT MAPING DB PLC 2"."P-501 B EDI FEED PUMP" )
      Coil( "P-501 B EDI FEED PUMP" )
   END_RUNG
   // the same network as SCL:
   "P-501 B EDI FEED PUMP" := "OUTPUT MAPING DB PLC 2"."P-501 B EDI FEED PUMP";
END_REGION

REGION Network 13: "P-501 C EDI FEED PUMP"
   RUNG wire#powerrail
      Contact( "OUTPUT MAPING DB PLC 2"."P-501 C EDI FEED PUMP" )
      Coil( "P-501 C EDI FEED PUMP" )
   END_RUNG
   // the same network as SCL:
   "P-501 C EDI FEED PUMP" := "OUTPUT MAPING DB PLC 2"."P-501 C EDI FEED PUMP";
END_REGION

REGION Network 14: "EDI 501"
   RUNG wire#powerrail
      Contact( "OUTPUT MAPING DB PLC 2"."EDI 501" )
      Coil( "EDI 501" )
   END_RUNG
   // the same network as SCL:
   "EDI 501" := "OUTPUT MAPING DB PLC 2"."EDI 501";
END_REGION

REGION Network 15: "EDI 502"
   RUNG wire#powerrail
      Contact( "OUTPUT MAPING DB PLC 2"."EDI 502" )
      Coil( "EDI 502" )
   END_RUNG
   // the same network as SCL:
   "EDI 502" := "OUTPUT MAPING DB PLC 2"."EDI 502";
END_REGION

REGION Network 16: "DP 703"
   RUNG wire#powerrail
      Contact( "OUTPUT MAPING DB PLC 2"."DP 703" )
      Coil( "DP 703" )
   END_RUNG
   // the same network as SCL:
   "DP 703" := "OUTPUT MAPING DB PLC 2"."DP 703";
END_REGION

REGION Network 17: "DP 704"
   RUNG wire#powerrail
      Contact( "OUTPUT MAPING DB PLC 2"."DP 704" )
      Coil( "DP 704" )
   END_RUNG
   // the same network as SCL:
   "DP 704" := "OUTPUT MAPING DB PLC 2"."DP 704";
END_REGION

REGION Network 18: "DP 705"
   RUNG wire#powerrail
      Contact( "OUTPUT MAPING DB PLC 2"."DP 705" )
      Coil( "DP 705" )
   END_RUNG
   // the same network as SCL:
   "DP 705" := "OUTPUT MAPING DB PLC 2"."DP 705";
END_REGION

REGION Network 19: "ABV 301"
   RUNG wire#powerrail
      Contact( "OUTPUT MAPING DB PLC 2"."ABV 301" )
      Coil( "ABV 301" )
   END_RUNG
   // the same network as SCL:
   "ABV 301" := "OUTPUT MAPING DB PLC 2"."ABV 301";
END_REGION

REGION Network 20: "ABV 302"
   RUNG wire#powerrail
      Contact( "OUTPUT MAPING DB PLC 2"."ABV 302" )
      Coil( "ABV 302" )
   END_RUNG
   // the same network as SCL:
   "ABV 302" := "OUTPUT MAPING DB PLC 2"."ABV 302";
END_REGION

REGION Network 21: "AGLV-301"
   RUNG wire#powerrail
      Contact( "OUTPUT MAPING DB PLC 2"."AGLV-301" )
      Coil( "AGLV-301" )
   END_RUNG
   // the same network as SCL:
   "AGLV-301" := "OUTPUT MAPING DB PLC 2"."AGLV-301";
END_REGION

REGION Network 22: "AGLV-302"
   RUNG wire#powerrail
      Contact( "OUTPUT MAPING DB PLC 2"."AGLV-302" )
      Coil( "AGLV-302" )
   END_RUNG
   // the same network as SCL:
   "AGLV-302" := "OUTPUT MAPING DB PLC 2"."AGLV-302";
END_REGION

REGION Network 23: "AGLV-401"
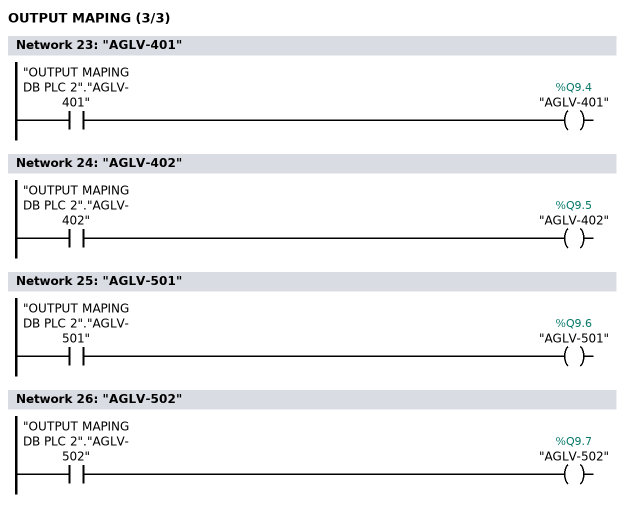
   RUNG wire#powerrail
      Contact( "OUTPUT MAPING DB PLC 2"."AGLV-401" )
      Coil( "AGLV-401" )
   END_RUNG
   // the same network as SCL:
   "AGLV-401" := "OUTPUT MAPING DB PLC 2"."AGLV-401";
END_REGION

REGION Network 24: "AGLV-402"
   RUNG wire#powerrail
      Contact( "OUTPUT MAPING DB PLC 2"."AGLV-402" )
      Coil( "AGLV-402" )
   END_RUNG
   // the same network as SCL:
   "AGLV-402" := "OUTPUT MAPING DB PLC 2"."AGLV-402";
END_REGION

REGION Network 25: "AGLV-501"
   RUNG wire#powerrail
      Contact( "OUTPUT MAPING DB PLC 2"."AGLV-501" )
      Coil( "AGLV-501" )
   END_RUNG
   // the same network as SCL:
   "AGLV-501" := "OUTPUT MAPING DB PLC 2"."AGLV-501";
END_REGION

REGION Network 26: "AGLV-502"
   RUNG wire#powerrail
      Contact( "OUTPUT MAPING DB PLC 2"."AGLV-502" )
      Coil( "AGLV-502" )
   END_RUNG
   // the same network as SCL:
   "AGLV-502" := "OUTPUT MAPING DB PLC 2"."AGLV-502";
END_REGION
END_FUNCTION

FUNCTION "MODE SELECTION" : Void   // FC3, LAD
{ S7_Optimized_Access := 'TRUE' }
// stored: SetENOAutomatically false
   VAR_TEMP   // added for the SCL form of the ladder/FBD networks
      _w1 : Bool;
   END_VAR
BEGIN

REGION Network 1: STANDBY \///////////////////////////////// RO-1 ///////////////////////////////////////////
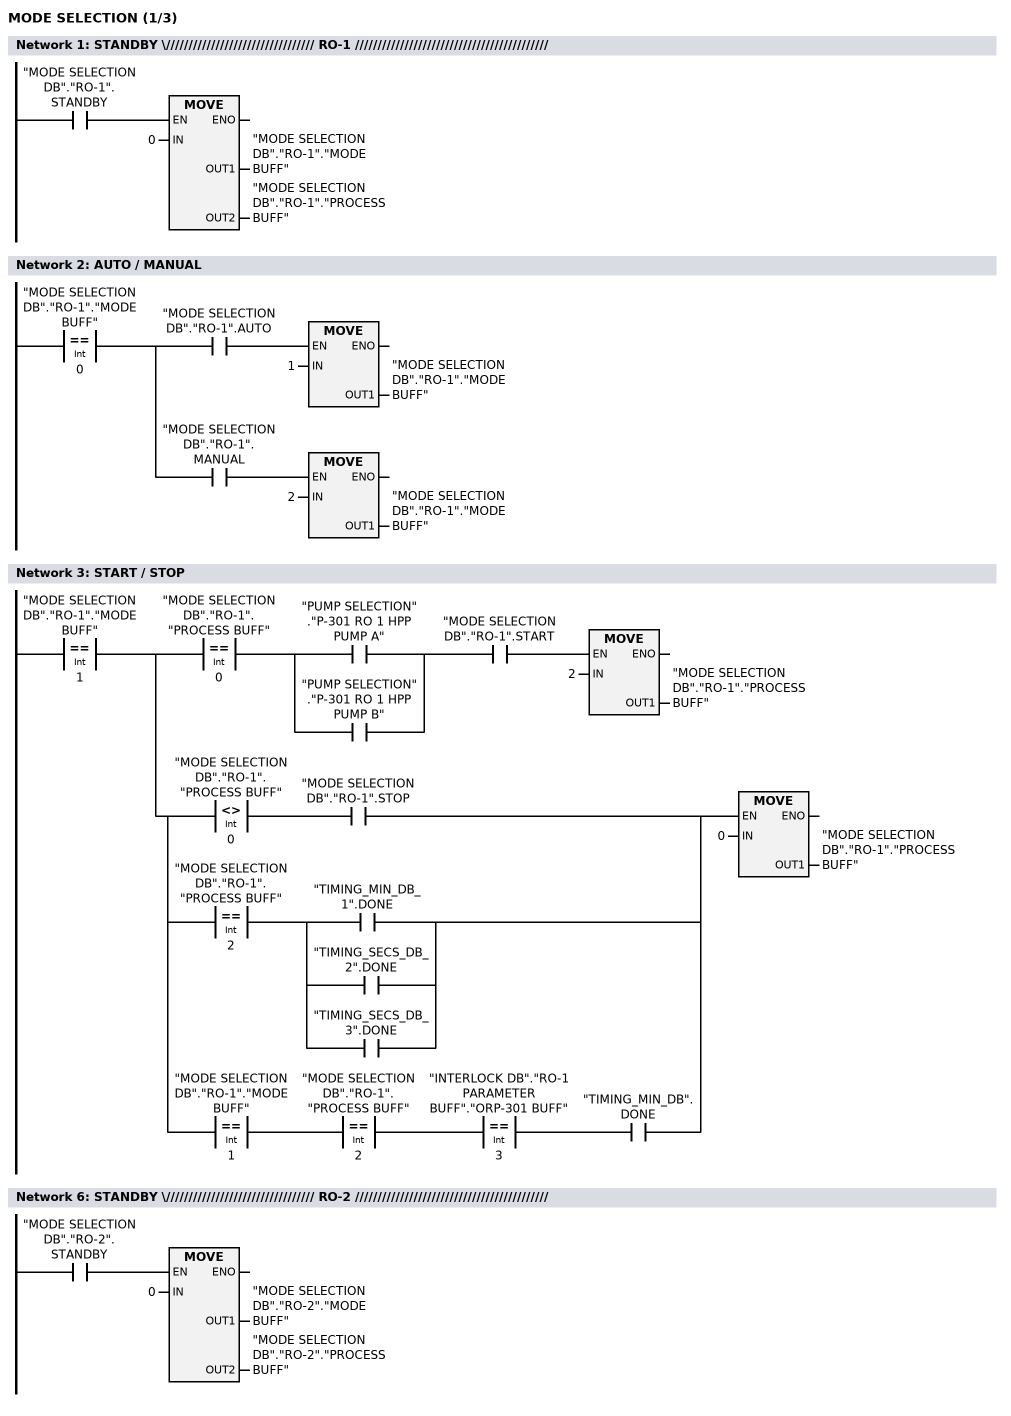
   RUNG wire#powerrail
      Contact( "MODE SELECTION DB"."RO-1".STANDBY )
      Move(in := 0, out1 => "MODE SELECTION DB"."RO-1"."MODE BUFF", out2 => "MODE SELECTION DB"."RO-1"."PROCESS BUFF")
   END_RUNG
   // the same network as SCL:
   IF "MODE SELECTION DB"."RO-1".STANDBY THEN
       "MODE SELECTION DB"."RO-1"."MODE BUFF" := 0;
       "MODE SELECTION DB"."RO-1"."PROCESS BUFF" := 0;
   END_IF;
END_REGION

REGION Network 2: AUTO / MANUAL
   RUNG wire#powerrail
      { S7_Templates := "SrcType := Int" } EQ_Contact(in1 := "MODE SELECTION DB"."RO-1"."MODE BUFF", in2 := 0)
      wire#w1
      Contact( "MODE SELECTION DB"."RO-1".AUTO )
      Move(in := 1, out1 => "MODE SELECTION DB"."RO-1"."MODE BUFF")
   END_RUNG
   RUNG wire#w1
      Contact( "MODE SELECTION DB"."RO-1".MANUAL )
      Move(in := 2, out1 => "MODE SELECTION DB"."RO-1"."MODE BUFF")
   END_RUNG
   // the same network as SCL:
   #_w1 := "MODE SELECTION DB"."RO-1"."MODE BUFF" = 0;
   IF #_w1 AND "MODE SELECTION DB"."RO-1".AUTO THEN "MODE SELECTION DB"."RO-1"."MODE BUFF" := 1; END_IF;
   IF #_w1 AND "MODE SELECTION DB"."RO-1".MANUAL THEN "MODE SELECTION DB"."RO-1"."MODE BUFF" := 2; END_IF;
END_REGION

REGION Network 3: START / STOP
   RUNG wire#powerrail
      { S7_Templates := "SrcType := Int" } EQ_Contact(in1 := "MODE SELECTION DB"."RO-1"."MODE BUFF", in2 := 1)
      wire#w1
      { S7_Templates := "SrcType := Int" } EQ_Contact(in1 := "MODE SELECTION DB"."RO-1"."PROCESS BUFF", in2 := 0)
      wire#w2
      Contact( "PUMP SELECTION"."P-301 RO 1 HPP PUMP A" )
      wire#w3
      Contact( "MODE SELECTION DB"."RO-1".START )
      Move(in := 2, out1 => "MODE SELECTION DB"."RO-1"."PROCESS BUFF")
   END_RUNG
   RUNG wire#w2
      Contact( "PUMP SELECTION"."P-301 RO 1 HPP PUMP B" )
   END_RUNG wire#w3
   RUNG wire#w1
      { S7_Templates := "SrcType := Int" } NE_Contact(in1 := "MODE SELECTION DB"."RO-1"."PROCESS BUFF", in2 := 0)
      Contact( "MODE SELECTION DB"."RO-1".STOP )
      wire#w4
      Move(in := 0, out1 => "MODE SELECTION DB"."RO-1"."PROCESS BUFF")
   END_RUNG
   RUNG wire#w1
      { S7_Templates := "SrcType := Int" } EQ_Contact(in1 := "MODE SELECTION DB"."RO-1"."PROCESS BUFF", in2 := 2)
      wire#w5
      Contact( "TIMING_MIN_DB_1".DONE )
   END_RUNG wire#w4
   RUNG wire#w5
      Contact( "TIMING_SECS_DB_2".DONE )
   END_RUNG wire#w4
   RUNG wire#w5
      Contact( "TIMING_SECS_DB_3".DONE )
   END_RUNG wire#w4
   RUNG wire#w1
      { S7_Templates := "SrcType := Int" } EQ_Contact(in1 := "MODE SELECTION DB"."RO-1"."MODE BUFF", in2 := 1)
      { S7_Templates := "SrcType := Int" } EQ_Contact(in1 := "MODE SELECTION DB"."RO-1"."PROCESS BUFF", in2 := 2)
      { S7_Templates := "SrcType := Int" } EQ_Contact(in1 := "INTERLOCK DB"."RO-1 PARAMETER BUFF"."ORP-301 BUFF", in2 := 3)
      Contact( "TIMING_MIN_DB".DONE )
   END_RUNG wire#w4
   // the same network as SCL:
   #_w1 := "MODE SELECTION DB"."RO-1"."MODE BUFF" = 1;
   IF #_w1 AND ("MODE SELECTION DB"."RO-1"."PROCESS BUFF" = 0) AND ("PUMP SELECTION"."P-301 RO 1 HPP PUMP A" OR "PUMP SELECTION"."P-301 RO 1 HPP PUMP B") AND "MODE SELECTION DB"."RO-1".START THEN
       "MODE SELECTION DB"."RO-1"."PROCESS BUFF" := 2;
   END_IF;
   IF #_w1 AND ((("MODE SELECTION DB"."RO-1"."PROCESS BUFF" <> 0) AND "MODE SELECTION DB"."RO-1".STOP) OR (("MODE SELECTION DB"."RO-1"."PROCESS BUFF" = 2) AND ("TIMING_MIN_DB_1".DONE OR "TIMING_SECS_DB_2".DONE OR "TIMING_SECS_DB_3".DONE)) OR (("MODE SELECTION DB"."RO-1"."MODE BUFF" = 1) AND ("MODE SELECTION DB"."RO-1"."PROCESS BUFF" = 2) AND ("INTERLOCK DB"."RO-1 PARAMETER BUFF"."ORP-301 BUFF" = 3) AND "TIMING_MIN_DB".DONE)) THEN
       "MODE SELECTION DB"."RO-1"."PROCESS BUFF" := 0;
   END_IF;
END_REGION

REGION Network 6: STANDBY \///////////////////////////////// RO-2 ///////////////////////////////////////////
   RUNG wire#powerrail
      Contact( "MODE SELECTION DB"."RO-2".STANDBY )
      Move(in := 0, out1 => "MODE SELECTION DB"."RO-2"."MODE BUFF", out2 => "MODE SELECTION DB"."RO-2"."PROCESS BUFF")
   END_RUNG
   // the same network as SCL:
   IF "MODE SELECTION DB"."RO-2".STANDBY THEN
       "MODE SELECTION DB"."RO-2"."MODE BUFF" := 0;
       "MODE SELECTION DB"."RO-2"."PROCESS BUFF" := 0;
   END_IF;
END_REGION

REGION Network 7: AUTO / MANUAL
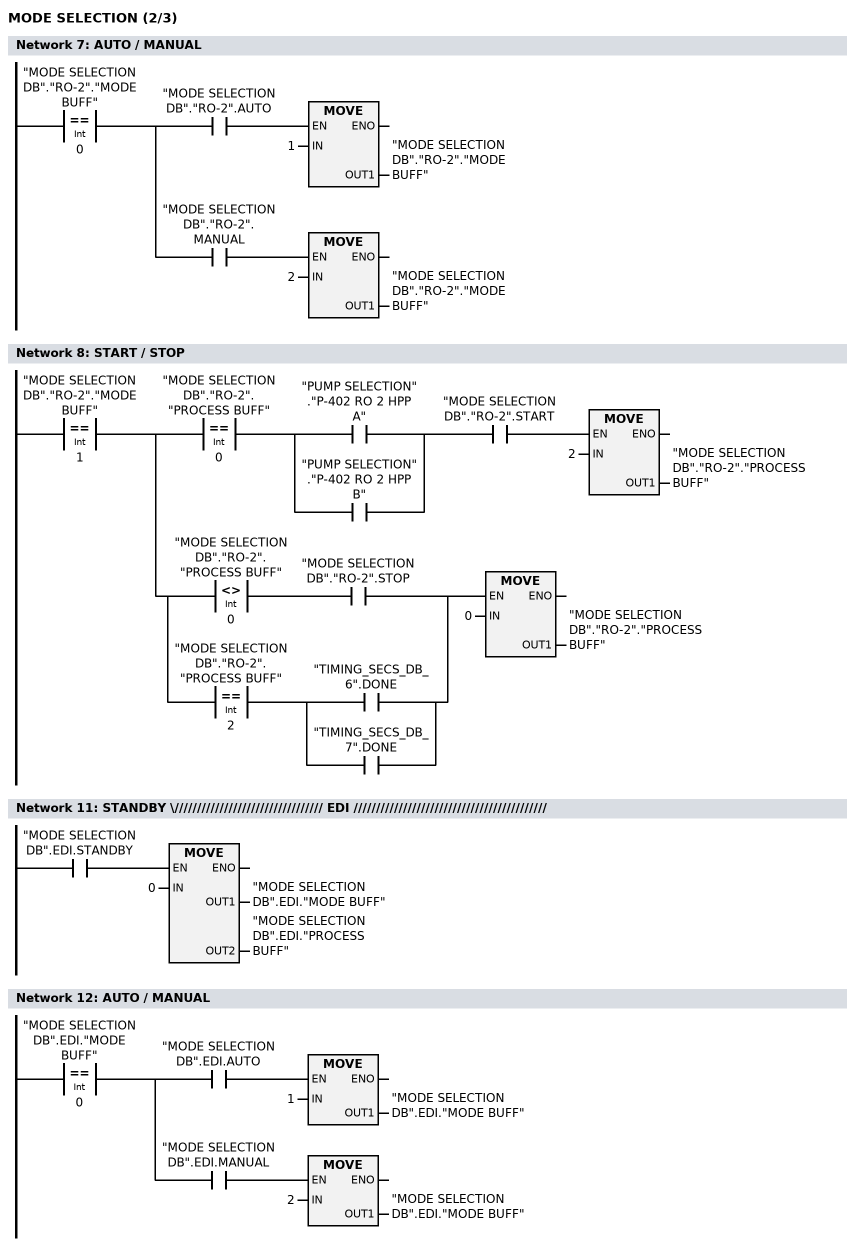
   RUNG wire#powerrail
      { S7_Templates := "SrcType := Int" } EQ_Contact(in1 := "MODE SELECTION DB"."RO-2"."MODE BUFF", in2 := 0)
      wire#w1
      Contact( "MODE SELECTION DB"."RO-2".AUTO )
      Move(in := 1, out1 => "MODE SELECTION DB"."RO-2"."MODE BUFF")
   END_RUNG
   RUNG wire#w1
      Contact( "MODE SELECTION DB"."RO-2".MANUAL )
      Move(in := 2, out1 => "MODE SELECTION DB"."RO-2"."MODE BUFF")
   END_RUNG
   // the same network as SCL:
   #_w1 := "MODE SELECTION DB"."RO-2"."MODE BUFF" = 0;
   IF #_w1 AND "MODE SELECTION DB"."RO-2".AUTO THEN "MODE SELECTION DB"."RO-2"."MODE BUFF" := 1; END_IF;
   IF #_w1 AND "MODE SELECTION DB"."RO-2".MANUAL THEN "MODE SELECTION DB"."RO-2"."MODE BUFF" := 2; END_IF;
END_REGION

REGION Network 8: START / STOP
   RUNG wire#powerrail
      { S7_Templates := "SrcType := Int" } EQ_Contact(in1 := "MODE SELECTION DB"."RO-2"."MODE BUFF", in2 := 1)
      wire#w1
      { S7_Templates := "SrcType := Int" } EQ_Contact(in1 := "MODE SELECTION DB"."RO-2"."PROCESS BUFF", in2 := 0)
      wire#w2
      Contact( "PUMP SELECTION"."P-402 RO 2 HPP A" )
      wire#w3
      Contact( "MODE SELECTION DB"."RO-2".START )
      Move(in := 2, out1 => "MODE SELECTION DB"."RO-2"."PROCESS BUFF")
   END_RUNG
   RUNG wire#w2
      Contact( "PUMP SELECTION"."P-402 RO 2 HPP B" )
   END_RUNG wire#w3
   RUNG wire#w1
      { S7_Templates := "SrcType := Int" } NE_Contact(in1 := "MODE SELECTION DB"."RO-2"."PROCESS BUFF", in2 := 0)
      Contact( "MODE SELECTION DB"."RO-2".STOP )
      wire#w4
      Move(in := 0, out1 => "MODE SELECTION DB"."RO-2"."PROCESS BUFF")
   END_RUNG
   RUNG wire#w1
      { S7_Templates := "SrcType := Int" } EQ_Contact(in1 := "MODE SELECTION DB"."RO-2"."PROCESS BUFF", in2 := 2)
      wire#w5
      Contact( "TIMING_SECS_DB_6".DONE )
   END_RUNG wire#w4
   RUNG wire#w5
      Contact( "TIMING_SECS_DB_7".DONE )
   END_RUNG wire#w4
   // the same network as SCL:
   #_w1 := "MODE SELECTION DB"."RO-2"."MODE BUFF" = 1;
   IF #_w1 AND ("MODE SELECTION DB"."RO-2"."PROCESS BUFF" = 0) AND ("PUMP SELECTION"."P-402 RO 2 HPP A" OR "PUMP SELECTION"."P-402 RO 2 HPP B") AND "MODE SELECTION DB"."RO-2".START THEN
       "MODE SELECTION DB"."RO-2"."PROCESS BUFF" := 2;
   END_IF;
   IF #_w1 AND ((("MODE SELECTION DB"."RO-2"."PROCESS BUFF" <> 0) AND "MODE SELECTION DB"."RO-2".STOP) OR (("MODE SELECTION DB"."RO-2"."PROCESS BUFF" = 2) AND ("TIMING_SECS_DB_6".DONE OR "TIMING_SECS_DB_7".DONE))) THEN
       "MODE SELECTION DB"."RO-2"."PROCESS BUFF" := 0;
   END_IF;
END_REGION

REGION Network 11: STANDBY \///////////////////////////////// EDI ///////////////////////////////////////////
   RUNG wire#powerrail
      Contact( "MODE SELECTION DB".EDI.STANDBY )
      Move(in := 0, out1 => "MODE SELECTION DB".EDI."MODE BUFF", out2 => "MODE SELECTION DB".EDI."PROCESS BUFF")
   END_RUNG
   // the same network as SCL:
   IF "MODE SELECTION DB".EDI.STANDBY THEN
       "MODE SELECTION DB".EDI."MODE BUFF" := 0;
       "MODE SELECTION DB".EDI."PROCESS BUFF" := 0;
   END_IF;
END_REGION

REGION Network 12: AUTO / MANUAL
   RUNG wire#powerrail
      { S7_Templates := "SrcType := Int" } EQ_Contact(in1 := "MODE SELECTION DB".EDI."MODE BUFF", in2 := 0)
      wire#w1
      Contact( "MODE SELECTION DB".EDI.AUTO )
      Move(in := 1, out1 => "MODE SELECTION DB".EDI."MODE BUFF")
   END_RUNG
   RUNG wire#w1
      Contact( "MODE SELECTION DB".EDI.MANUAL )
      Move(in := 2, out1 => "MODE SELECTION DB".EDI."MODE BUFF")
   END_RUNG
   // the same network as SCL:
   #_w1 := "MODE SELECTION DB".EDI."MODE BUFF" = 0;
   IF #_w1 AND "MODE SELECTION DB".EDI.AUTO THEN "MODE SELECTION DB".EDI."MODE BUFF" := 1; END_IF;
   IF #_w1 AND "MODE SELECTION DB".EDI.MANUAL THEN "MODE SELECTION DB".EDI."MODE BUFF" := 2; END_IF;
END_REGION

REGION Network 13: START / STOP
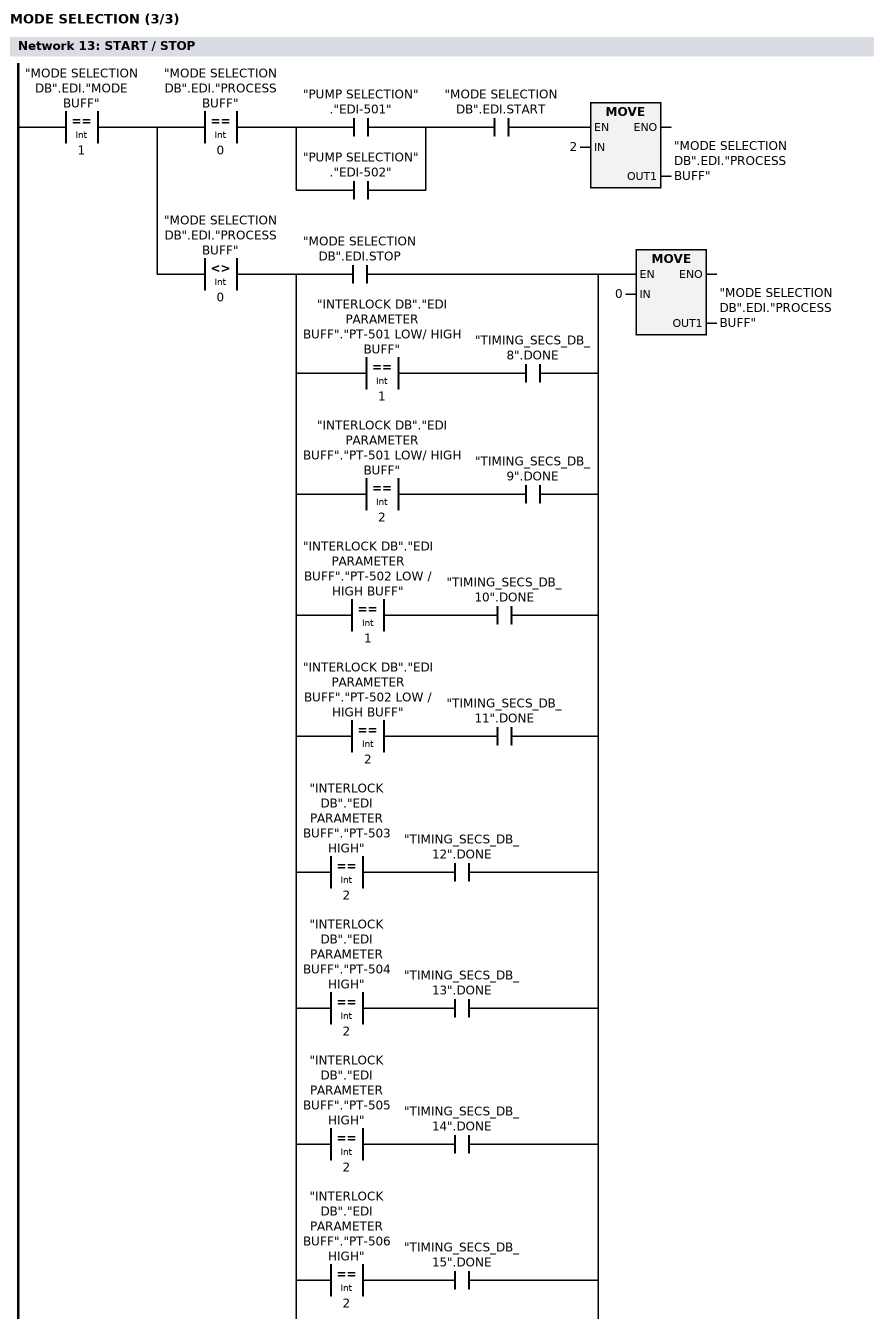
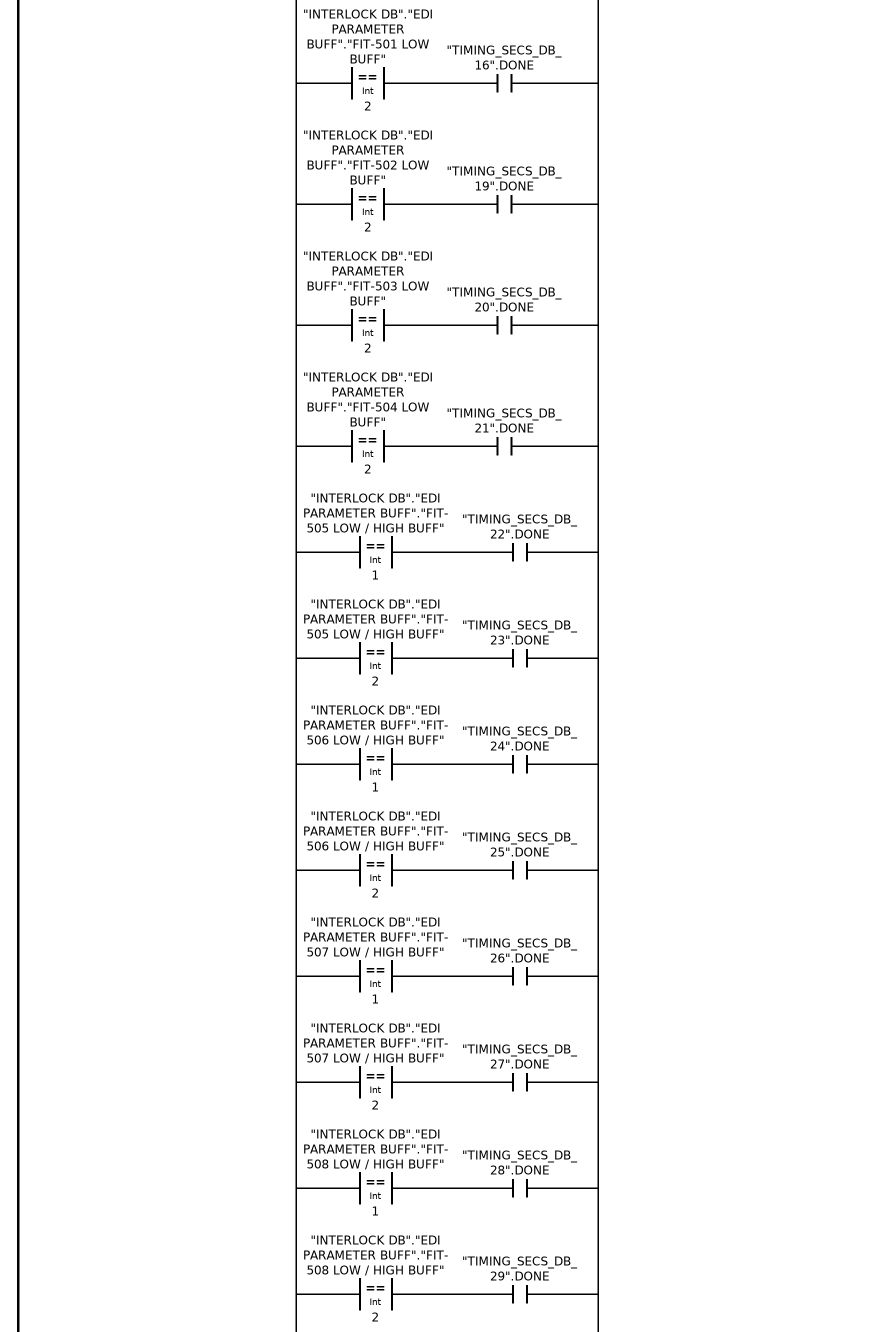
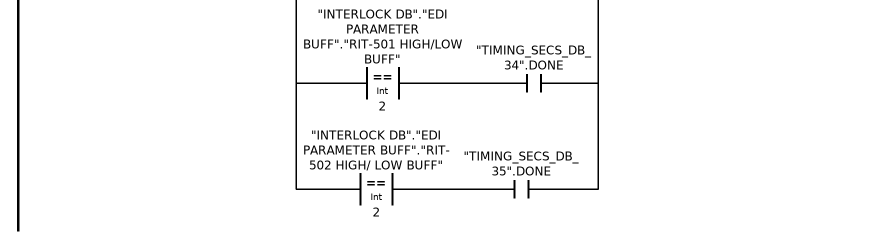
   RUNG wire#powerrail
      { S7_Templates := "SrcType := Int" } EQ_Contact(in1 := "MODE SELECTION DB".EDI."MODE BUFF", in2 := 1)
      wire#w1
      { S7_Templates := "SrcType := Int" } EQ_Contact(in1 := "MODE SELECTION DB".EDI."PROCESS BUFF", in2 := 0)
      wire#w2
      Contact( "PUMP SELECTION"."EDI-501" )
      wire#w3
      Contact( "MODE SELECTION DB".EDI.START )
      Move(in := 2, out1 => "MODE SELECTION DB".EDI."PROCESS BUFF")
   END_RUNG
   RUNG wire#w2
      Contact( "PUMP SELECTION"."EDI-502" )
   END_RUNG wire#w3
   RUNG wire#w1
      { S7_Templates := "SrcType := Int" } NE_Contact(in1 := "MODE SELECTION DB".EDI."PROCESS BUFF", in2 := 0)
      wire#w4
      Contact( "MODE SELECTION DB".EDI.STOP )
      wire#w5
      Move(in := 0, out1 => "MODE SELECTION DB".EDI."PROCESS BUFF")
   END_RUNG
   RUNG wire#w4
      { S7_Templates := "SrcType := Int" } EQ_Contact(in1 := "INTERLOCK DB"."EDI PARAMETER BUFF"."PT-501 LOW/ HIGH BUFF", in2 := 1)
      Contact( "TIMING_SECS_DB_8".DONE )
   END_RUNG wire#w5
   RUNG wire#w4
      { S7_Templates := "SrcType := Int" } EQ_Contact(in1 := "INTERLOCK DB"."EDI PARAMETER BUFF"."PT-501 LOW/ HIGH BUFF", in2 := 2)
      Contact( "TIMING_SECS_DB_9".DONE )
   END_RUNG wire#w5
   RUNG wire#w4
      { S7_Templates := "SrcType := Int" } EQ_Contact(in1 := "INTERLOCK DB"."EDI PARAMETER BUFF"."PT-502 LOW / HIGH BUFF", in2 := 1)
      Contact( "TIMING_SECS_DB_10".DONE )
   END_RUNG wire#w5
   RUNG wire#w4
      { S7_Templates := "SrcType := Int" } EQ_Contact(in1 := "INTERLOCK DB"."EDI PARAMETER BUFF"."PT-502 LOW / HIGH BUFF", in2 := 2)
      Contact( "TIMING_SECS_DB_11".DONE )
   END_RUNG wire#w5
   RUNG wire#w4
      { S7_Templates := "SrcType := Int" } EQ_Contact(in1 := "INTERLOCK DB"."EDI PARAMETER BUFF"."PT-503 HIGH", in2 := 2)
      Contact( "TIMING_SECS_DB_12".DONE )
   END_RUNG wire#w5
   RUNG wire#w4
      { S7_Templates := "SrcType := Int" } EQ_Contact(in1 := "INTERLOCK DB"."EDI PARAMETER BUFF"."PT-504 HIGH", in2 := 2)
      Contact( "TIMING_SECS_DB_13".DONE )
   END_RUNG wire#w5
   RUNG wire#w4
      { S7_Templates := "SrcType := Int" } EQ_Contact(in1 := "INTERLOCK DB"."EDI PARAMETER BUFF"."PT-505 HIGH", in2 := 2)
      Contact( "TIMING_SECS_DB_14".DONE )
   END_RUNG wire#w5
   RUNG wire#w4
      { S7_Templates := "SrcType := Int" } EQ_Contact(in1 := "INTERLOCK DB"."EDI PARAMETER BUFF"."PT-506 HIGH", in2 := 2)
      Contact( "TIMING_SECS_DB_15".DONE )
   END_RUNG wire#w5
   RUNG wire#w4
      { S7_Templates := "SrcType := Int" } EQ_Contact(in1 := "INTERLOCK DB"."EDI PARAMETER BUFF"."FIT-501 LOW BUFF", in2 := 2)
      Contact( "TIMING_SECS_DB_16".DONE )
   END_RUNG wire#w5
   RUNG wire#w4
      { S7_Templates := "SrcType := Int" } EQ_Contact(in1 := "INTERLOCK DB"."EDI PARAMETER BUFF"."FIT-502 LOW  BUFF", in2 := 2)
      Contact( "TIMING_SECS_DB_19".DONE )
   END_RUNG wire#w5
   RUNG wire#w4
      { S7_Templates := "SrcType := Int" } EQ_Contact(in1 := "INTERLOCK DB"."EDI PARAMETER BUFF"."FIT-503 LOW BUFF", in2 := 2)
      Contact( "TIMING_SECS_DB_20".DONE )
   END_RUNG wire#w5
   RUNG wire#w4
      { S7_Templates := "SrcType := Int" } EQ_Contact(in1 := "INTERLOCK DB"."EDI PARAMETER BUFF"."FIT-504 LOW BUFF", in2 := 2)
      Contact( "TIMING_SECS_DB_21".DONE )
   END_RUNG wire#w5
   RUNG wire#w4
      { S7_Templates := "SrcType := Int" } EQ_Contact(in1 := "INTERLOCK DB"."EDI PARAMETER BUFF"."FIT-505 LOW / HIGH BUFF", in2 := 1)
      Contact( "TIMING_SECS_DB_22".DONE )
   END_RUNG wire#w5
   RUNG wire#w4
      { S7_Templates := "SrcType := Int" } EQ_Contact(in1 := "INTERLOCK DB"."EDI PARAMETER BUFF"."FIT-505 LOW / HIGH BUFF", in2 := 2)
      Contact( "TIMING_SECS_DB_23".DONE )
   END_RUNG wire#w5
   RUNG wire#w4
      { S7_Templates := "SrcType := Int" } EQ_Contact(in1 := "INTERLOCK DB"."EDI PARAMETER BUFF"."FIT-506 LOW / HIGH BUFF", in2 := 1)
      Contact( "TIMING_SECS_DB_24".DONE )
   END_RUNG wire#w5
   RUNG wire#w4
      { S7_Templates := "SrcType := Int" } EQ_Contact(in1 := "INTERLOCK DB"."EDI PARAMETER BUFF"."FIT-506 LOW / HIGH BUFF", in2 := 2)
      Contact( "TIMING_SECS_DB_25".DONE )
   END_RUNG wire#w5
   RUNG wire#w4
      { S7_Templates := "SrcType := Int" } EQ_Contact(in1 := "INTERLOCK DB"."EDI PARAMETER BUFF"."FIT-507 LOW / HIGH BUFF", in2 := 1)
      Contact( "TIMING_SECS_DB_26".DONE )
   END_RUNG wire#w5
   RUNG wire#w4
      { S7_Templates := "SrcType := Int" } EQ_Contact(in1 := "INTERLOCK DB"."EDI PARAMETER BUFF"."FIT-507 LOW / HIGH BUFF", in2 := 2)
      Contact( "TIMING_SECS_DB_27".DONE )
   END_RUNG wire#w5
   RUNG wire#w4
      { S7_Templates := "SrcType := Int" } EQ_Contact(in1 := "INTERLOCK DB"."EDI PARAMETER BUFF"."FIT-508 LOW / HIGH BUFF", in2 := 1)
      Contact( "TIMING_SECS_DB_28".DONE )
   END_RUNG wire#w5
   RUNG wire#w4
      { S7_Templates := "SrcType := Int" } EQ_Contact(in1 := "INTERLOCK DB"."EDI PARAMETER BUFF"."FIT-508 LOW / HIGH BUFF", in2 := 2)
      Contact( "TIMING_SECS_DB_29".DONE )
   END_RUNG wire#w5
   RUNG wire#w4
      { S7_Templates := "SrcType := Int" } EQ_Contact(in1 := "INTERLOCK DB"."EDI PARAMETER BUFF"."RIT-501 HIGH/LOW BUFF", in2 := 2)
      Contact( "TIMING_SECS_DB_34".DONE )
   END_RUNG wire#w5
   RUNG wire#w4
      { S7_Templates := "SrcType := Int" } EQ_Contact(in1 := "INTERLOCK DB"."EDI PARAMETER BUFF"."RIT-502 HIGH/ LOW BUFF", in2 := 2)
      Contact( "TIMING_SECS_DB_35".DONE )
   END_RUNG wire#w5
   // the same network as SCL:
   #_w1 := "MODE SELECTION DB".EDI."MODE BUFF" = 1;
   IF #_w1 AND ("MODE SELECTION DB".EDI."PROCESS BUFF" = 0) AND ("PUMP SELECTION"."EDI-501" OR "PUMP SELECTION"."EDI-502") AND "MODE SELECTION DB".EDI.START THEN
       "MODE SELECTION DB".EDI."PROCESS BUFF" := 2;
   END_IF;
   IF #_w1 AND ("MODE SELECTION DB".EDI."PROCESS BUFF" <> 0) AND ("MODE SELECTION DB".EDI.STOP OR (("INTERLOCK DB"."EDI PARAMETER BUFF"."PT-501 LOW/ HIGH BUFF" = 1) AND "TIMING_SECS_DB_8".DONE) OR (("INTERLOCK DB"."EDI PARAMETER BUFF"."PT-501 LOW/ HIGH BUFF" = 2) AND "TIMING_SECS_DB_9".DONE) OR (("INTERLOCK DB"."EDI PARAMETER BUFF"."PT-502 LOW / HIGH BUFF" = 1) AND "TIMING_SECS_DB_10".DONE) OR (("INTERLOCK DB"."EDI PARAMETER BUFF"."PT-502 LOW / HIGH BUFF" = 2) AND "TIMING_SECS_DB_11".DONE) OR (("INTERLOCK DB"."EDI PARAMETER BUFF"."PT-503 HIGH" = 2) AND "TIMING_SECS_DB_12".DONE) OR (("INTERLOCK DB"."EDI PARAMETER BUFF"."PT-504 HIGH" = 2) AND "TIMING_SECS_DB_13".DONE) OR (("INTERLOCK DB"."EDI PARAMETER BUFF"."PT-505 HIGH" = 2) AND "TIMING_SECS_DB_14".DONE) OR (("INTERLOCK DB"."EDI PARAMETER BUFF"."PT-506 HIGH" = 2) AND "TIMING_SECS_DB_15".DONE) OR (("INTERLOCK DB"."EDI PARAMETER BUFF"."FIT-501 LOW BUFF" = 2) AND "TIMING_SECS_DB_16".DONE) OR (("INTERLOCK DB"."EDI PARAMETER BUFF"."FIT-502 LOW  BUFF" = 2) AND "TIMING_SECS_DB_19".DONE) OR (("INTERLOCK DB"."EDI PARAMETER BUFF"."FIT-503 LOW BUFF" = 2) AND "TIMING_SECS_DB_20".DONE) OR (("INTERLOCK DB"."EDI PARAMETER BUFF"."FIT-504 LOW BUFF" = 2) AND "TIMING_SECS_DB_21".DONE) OR (("INTERLOCK DB"."EDI PARAMETER BUFF"."FIT-505 LOW / HIGH BUFF" = 1) AND "TIMING_SECS_DB_22".DONE) OR (("INTERLOCK DB"."EDI PARAMETER BUFF"."FIT-505 LOW / HIGH BUFF" = 2) AND "TIMING_SECS_DB_23".DONE) OR (("INTERLOCK DB"."EDI PARAMETER BUFF"."FIT-506 LOW / HIGH BUFF" = 1) AND "TIMING_SECS_DB_24".DONE) OR (("INTERLOCK DB"."EDI PARAMETER BUFF"."FIT-506 LOW / HIGH BUFF" = 2) AND "TIMING_SECS_DB_25".DONE) OR (("INTERLOCK DB"."EDI PARAMETER BUFF"."FIT-507 LOW / HIGH BUFF" = 1) AND "TIMING_SECS_DB_26".DONE) OR (("INTERLOCK DB"."EDI PARAMETER BUFF"."FIT-507 LOW / HIGH BUFF" = 2) AND "TIMING_SECS_DB_27".DONE) OR (("INTERLOCK DB"."EDI PARAMETER BUFF"."FIT-508 LOW / HIGH BUFF" = 1) AND "TIMING_SECS_DB_28".DONE) OR (("INTERLOCK DB"."EDI PARAMETER BUFF"."FIT-508 LOW / HIGH BUFF" = 2) AND "TIMING_SECS_DB_29".DONE) OR (("INTERLOCK DB"."EDI PARAMETER BUFF"."RIT-501 HIGH/LOW BUFF" = 2) AND "TIMING_SECS_DB_34".DONE) OR (("INTERLOCK DB"."EDI PARAMETER BUFF"."RIT-502 HIGH/ LOW BUFF" = 2) AND "TIMING_SECS_DB_35".DONE)) THEN
       "MODE SELECTION DB".EDI."PROCESS BUFF" := 0;
   END_IF;
END_REGION
END_FUNCTION

FUNCTION "FLUSHING VAVLE" : Void
{ S7_Optimized_Access := 'TRUE' }
VERSION : 0.1

BEGIN
	"ABV 301_FLUSH"("SUBOUTPUT VALVE":="OUTPUT MAPING DB PLC 2"."ABV 301",
	                "OPEN FEEDBACK":="INPUT MAPING DB"."ABFV-301 FEED BACK OPEN",
	                "CLOSE FEEDBACK":="INPUT MAPING DB"."ABFV-301 FEED BACK CLOSE",
	                "OPEN OUTPUT VAVLE"=>"FLUSHING VAVLE DB"."ABV 301",
	                "CLOSE OUTPUT VAVLE"=>"FLUSHING VAVLE DB"."ABV 301 CLOSE VALVE");
	
	"ABV 302_FLUSH"("SUBOUTPUT VALVE":="OUTPUT MAPING DB PLC 2"."ABV 302",
	                "OPEN FEEDBACK":="INPUT MAPING DB"."ABFV-302 OPEN FEED BACK",
	                "CLOSE FEEDBACK":="INPUT MAPING DB"."ABFV-302 CLOSE FEED BACK",
	                    "OPEN OUTPUT VAVLE"=>"FLUSHING VAVLE DB"."ABV 302",
	                "CLOSE OUTPUT VAVLE"=>"FLUSHING VAVLE DB"."ABV 302 CLOSE VALVE");
	
	"AGLV-301_FLUSH"("SUBOUTPUT VALVE":="OUTPUT MAPING DB PLC 2"."AGLV-301",
	                 "OPEN FEEDBACK":="INPUT MAPING DB"."AGLV-301 OPEN FEED BACK",
	                 "CLOSE FEEDBACK":="INPUT MAPING DB"."AGLV-301 CLOSE FEED BACK",
	                 "OPEN OUTPUT VAVLE"=>"FLUSHING VAVLE DB"."AGLV-301",
	                 "CLOSE OUTPUT VAVLE"=>"FLUSHING VAVLE DB"."AGLV 301 CLOSE VALVE");
	
	"AGLV-302_FLUSH"("SUBOUTPUT VALVE":="OUTPUT MAPING DB PLC 2"."AGLV-302",
	                 "OPEN FEEDBACK":="INPUT MAPING DB"."AGLV-302 OPEN FEED BACK",
	                 "CLOSE FEEDBACK":="INPUT MAPING DB"."AGLV-302 CLOSE FEED BACK",
	                 "OPEN OUTPUT VAVLE"=>"FLUSHING VAVLE DB"."AGLV-302",
	                 "CLOSE OUTPUT VAVLE"=>"FLUSHING VAVLE DB"."AGLV 302 CLOSE VALVE");
	
	"AGLV-401_FLUSH"("SUBOUTPUT VALVE":="OUTPUT MAPING DB PLC 2"."AGLV-401",
	                 "OPEN FEEDBACK":="INPUT MAPING DB"."AGLV-401 OPEN FEED BACK",
	                 "CLOSE FEEDBACK":="INPUT MAPING DB"."AGLV-401 CLOSE FEED BACK",
	                 "OPEN OUTPUT VAVLE"=>"FLUSHING VAVLE DB"."AGLV-401",
	                 "CLOSE OUTPUT VAVLE"=>"FLUSHING VAVLE DB"."AGLV 401 CLOSE VALVE");
	
	
	"AGLV-402_FLUSH"("SUBOUTPUT VALVE":="OUTPUT MAPING DB PLC 2"."AGLV-402",
	                 "OPEN FEEDBACK":="INPUT MAPING DB"."AGLV-402 OPEN FEED BACK",
	                 "CLOSE FEEDBACK":="INPUT MAPING DB"."AGLV-402 CLOSE FEED BACK",
	                 "OPEN OUTPUT VAVLE"=>"FLUSHING VAVLE DB"."AGLV-402",
	                 "CLOSE OUTPUT VAVLE"=>"FLUSHING VAVLE DB"."AGLV-402 CLOSE VALVE");
	
	"ABFV 501_FLUSH"("SUBOUTPUT VALVE":="OUTPUT MAPING DB PLC 2"."AGLV-501",
	                 "OPEN FEEDBACK":="INPUT MAPING DB"."AGLV-501OPEN FEED BACK",
	                 "CLOSE FEEDBACK":="INPUT MAPING DB"."AGLV-501 CLOSE FEED BACK",
	                 "OPEN OUTPUT VAVLE"=>"FLUSHING VAVLE DB"."ABFV 501",
	                 "CLOSE OUTPUT VAVLE"=>"FLUSHING VAVLE DB"."ABFV 501 CLOSE VALVE");
	
	"ABFV 502_FLUSH"("SUBOUTPUT VALVE":="OUTPUT MAPING DB PLC 2"."AGLV-502",
	                 "OPEN FEEDBACK":="INPUT MAPING DB"."AGLV-502 OPEN FEED BACK",
	                 "CLOSE FEEDBACK":="INPUT MAPING DB"."AGLV-502 CLOSE FEED BACK",
	                 "OPEN OUTPUT VAVLE"=>"FLUSHING VAVLE DB"."ABFV 502",
	                 "CLOSE OUTPUT VAVLE"=>"FLUSHING VAVLE DB"."ABFV 502 CLOSE VALVE");
	
	
	
	
	
	
	
	
	
	
	
	
	
	
	
	
	
	
END_FUNCTION

FUNCTION "INTERLOCK" : Void   // FC8, LAD
{ S7_Optimized_Access := 'TRUE' }
// stored: SetENOAutomatically false
   VAR_TEMP   // added for the SCL form of the ladder/FBD networks
      _w1 : Bool;
      _w2 : Bool;
   END_VAR
BEGIN

REGION Network 1: RO-1 RESET INTERLOCK
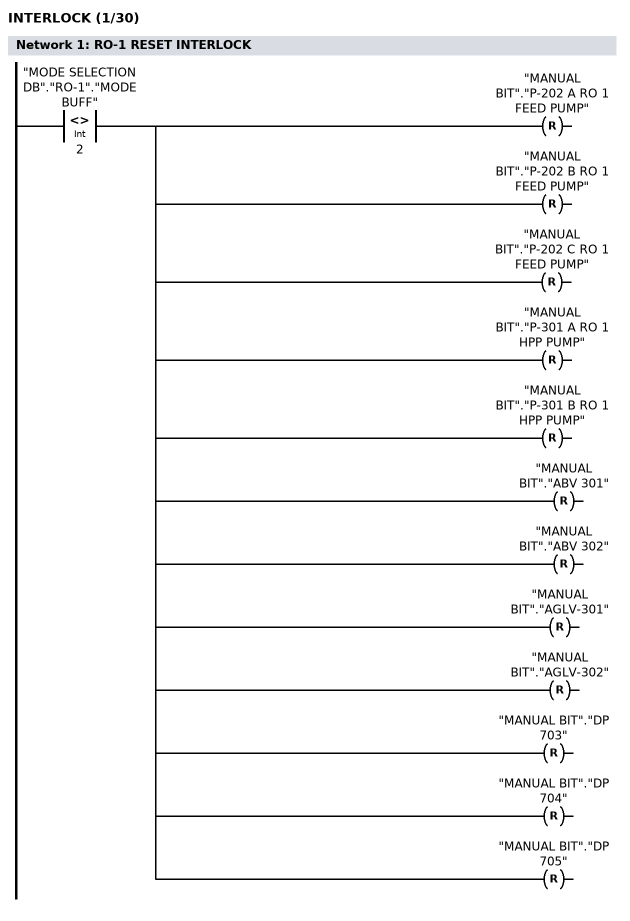
   RUNG wire#powerrail
      { S7_Templates := "SrcType := Int" } NE_Contact(in1 := "MODE SELECTION DB"."RO-1"."MODE BUFF", in2 := 2)
      wire#w1
      R_Coil( "MANUAL BIT"."P-202 A RO 1 FEED PUMP" )
   END_RUNG
   RUNG wire#w1
      R_Coil( "MANUAL BIT"."P-202 B RO 1 FEED PUMP" )
   END_RUNG
   RUNG wire#w1
      R_Coil( "MANUAL BIT"."P-202 C RO 1 FEED PUMP" )
   END_RUNG
   RUNG wire#w1
      R_Coil( "MANUAL BIT"."P-301 A RO 1 HPP PUMP" )
   END_RUNG
   RUNG wire#w1
      R_Coil( "MANUAL BIT"."P-301 B RO 1 HPP PUMP" )
   END_RUNG
   RUNG wire#w1
      R_Coil( "MANUAL BIT"."ABV 301" )
   END_RUNG
   RUNG wire#w1
      R_Coil( "MANUAL BIT"."ABV 302" )
   END_RUNG
   RUNG wire#w1
      R_Coil( "MANUAL BIT"."AGLV-301" )
   END_RUNG
   RUNG wire#w1
      R_Coil( "MANUAL BIT"."AGLV-302" )
   END_RUNG
   RUNG wire#w1
      R_Coil( "MANUAL BIT"."DP 703" )
   END_RUNG
   RUNG wire#w1
      R_Coil( "MANUAL BIT"."DP 704" )
   END_RUNG
   RUNG wire#w1
      R_Coil( "MANUAL BIT"."DP 705" )
   END_RUNG
   // the same network as SCL:
   IF "MODE SELECTION DB"."RO-1"."MODE BUFF" <> 2 THEN
       "MANUAL BIT"."P-202 A RO 1 FEED PUMP" := FALSE;
       "MANUAL BIT"."P-202 B RO 1 FEED PUMP" := FALSE;
       "MANUAL BIT"."P-202 C RO 1 FEED PUMP" := FALSE;
       "MANUAL BIT"."P-301 A RO 1 HPP PUMP" := FALSE;
       "MANUAL BIT"."P-301 B RO 1 HPP PUMP" := FALSE;
       "MANUAL BIT"."ABV 301" := FALSE;
       "MANUAL BIT"."ABV 302" := FALSE;
       "MANUAL BIT"."AGLV-301" := FALSE;
       "MANUAL BIT"."AGLV-302" := FALSE;
       "MANUAL BIT"."DP 703" := FALSE;
       "MANUAL BIT"."DP 704" := FALSE;
       "MANUAL BIT"."DP 705" := FALSE;
   END_IF;
END_REGION

REGION Network 2: RO-2 RESET INTERLOCK
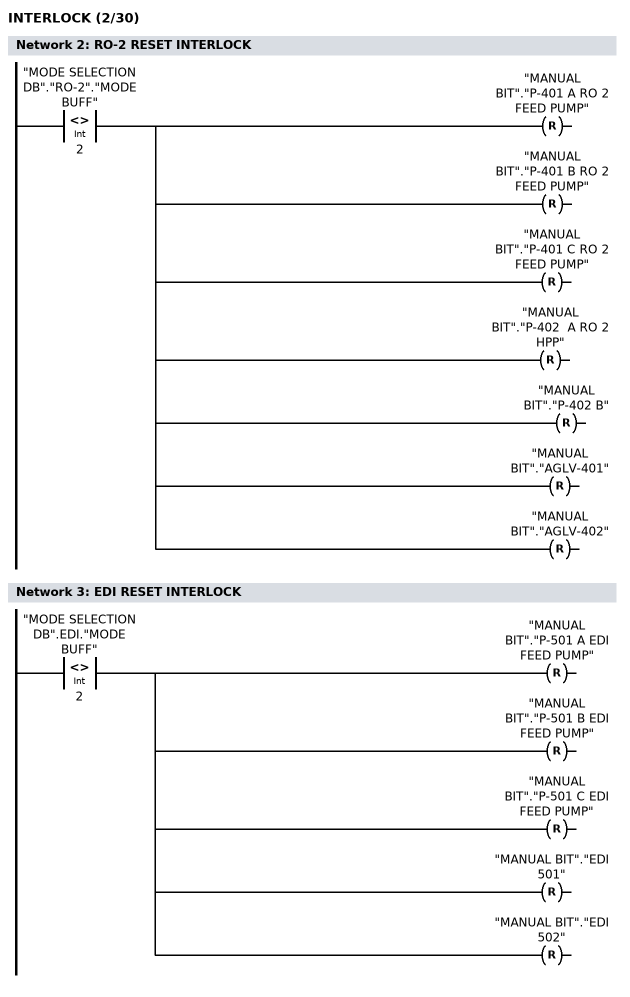
   RUNG wire#powerrail
      { S7_Templates := "SrcType := Int" } NE_Contact(in1 := "MODE SELECTION DB"."RO-2"."MODE BUFF", in2 := 2)
      wire#w1
      R_Coil( "MANUAL BIT"."P-401 A RO 2 FEED PUMP" )
   END_RUNG
   RUNG wire#w1
      R_Coil( "MANUAL BIT"."P-401 B RO 2 FEED PUMP" )
   END_RUNG
   RUNG wire#w1
      R_Coil( "MANUAL BIT"."P-401 C RO 2 FEED PUMP" )
   END_RUNG
   RUNG wire#w1
      R_Coil( "MANUAL BIT"."P-402  A RO 2 HPP" )
   END_RUNG
   RUNG wire#w1
      R_Coil( "MANUAL BIT"."P-402 B" )
   END_RUNG
   RUNG wire#w1
      R_Coil( "MANUAL BIT"."AGLV-401" )
   END_RUNG
   RUNG wire#w1
      R_Coil( "MANUAL BIT"."AGLV-402" )
   END_RUNG
   // the same network as SCL:
   IF "MODE SELECTION DB"."RO-2"."MODE BUFF" <> 2 THEN
       "MANUAL BIT"."P-401 A RO 2 FEED PUMP" := FALSE;
       "MANUAL BIT"."P-401 B RO 2 FEED PUMP" := FALSE;
       "MANUAL BIT"."P-401 C RO 2 FEED PUMP" := FALSE;
       "MANUAL BIT"."P-402  A RO 2 HPP" := FALSE;
       "MANUAL BIT"."P-402 B" := FALSE;
       "MANUAL BIT"."AGLV-401" := FALSE;
       "MANUAL BIT"."AGLV-402" := FALSE;
   END_IF;
END_REGION

REGION Network 3: EDI RESET INTERLOCK
   RUNG wire#powerrail
      { S7_Templates := "SrcType := Int" } NE_Contact(in1 := "MODE SELECTION DB".EDI."MODE BUFF", in2 := 2)
      wire#w1
      R_Coil( "MANUAL BIT"."P-501 A EDI FEED PUMP" )
   END_RUNG
   RUNG wire#w1
      R_Coil( "MANUAL BIT"."P-501 B EDI FEED PUMP" )
   END_RUNG
   RUNG wire#w1
      R_Coil( "MANUAL BIT"."P-501 C EDI FEED PUMP" )
   END_RUNG
   RUNG wire#w1
      R_Coil( "MANUAL BIT"."EDI 501" )
   END_RUNG
   RUNG wire#w1
      R_Coil( "MANUAL BIT"."EDI 502" )
   END_RUNG
   // the same network as SCL:
   IF "MODE SELECTION DB".EDI."MODE BUFF" <> 2 THEN
       "MANUAL BIT"."P-501 A EDI FEED PUMP" := FALSE;
       "MANUAL BIT"."P-501 B EDI FEED PUMP" := FALSE;
       "MANUAL BIT"."P-501 C EDI FEED PUMP" := FALSE;
       "MANUAL BIT"."EDI 501" := FALSE;
       "MANUAL BIT"."EDI 502" := FALSE;
   END_IF;
END_REGION

REGION Network 4: SELECTION PUMP INTERLOCK_
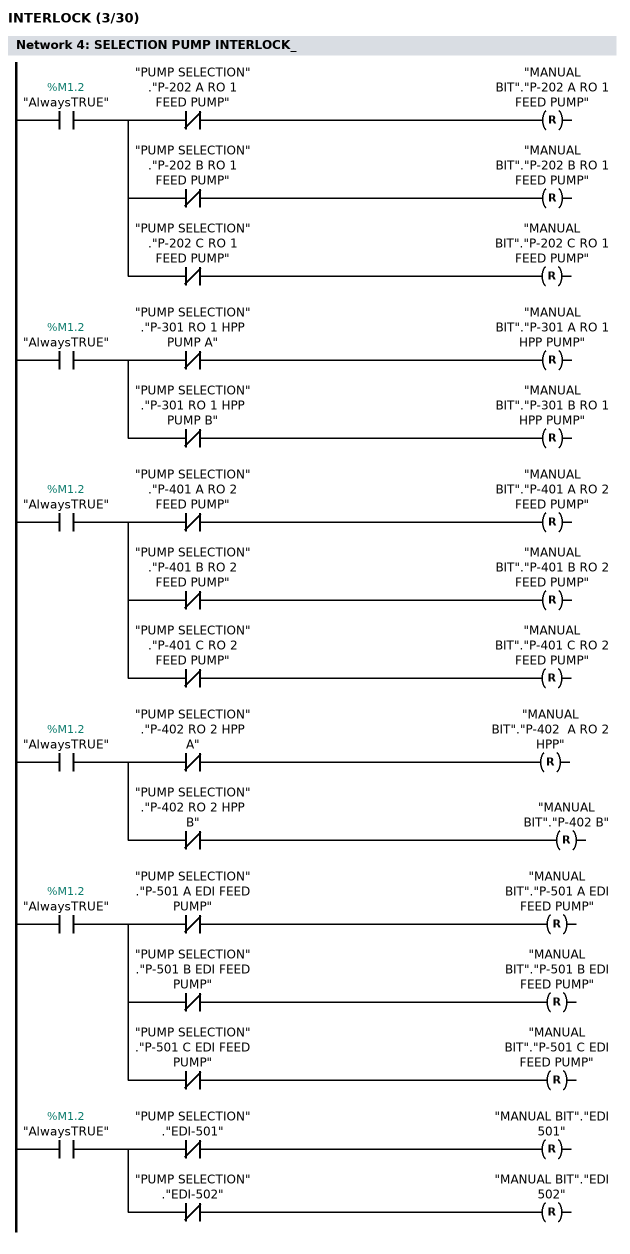
   RUNG wire#powerrail
      Contact( "AlwaysTRUE" )
      wire#w1
      I_Contact( "PUMP SELECTION"."P-202 A RO 1 FEED PUMP" )
      R_Coil( "MANUAL BIT"."P-202 A RO 1 FEED PUMP" )
   END_RUNG
   RUNG wire#w1
      I_Contact( "PUMP SELECTION"."P-202 B RO 1 FEED PUMP" )
      R_Coil( "MANUAL BIT"."P-202 B RO 1 FEED PUMP" )
   END_RUNG
   RUNG wire#w1
      I_Contact( "PUMP SELECTION"."P-202 C RO 1 FEED PUMP" )
      R_Coil( "MANUAL BIT"."P-202 C RO 1 FEED PUMP" )
   END_RUNG
   RUNG wire#powerrail
      Contact( "AlwaysTRUE" )
      wire#w2
      I_Contact( "PUMP SELECTION"."P-301 RO 1 HPP PUMP A" )
      R_Coil( "MANUAL BIT"."P-301 A RO 1 HPP PUMP" )
   END_RUNG
   RUNG wire#w2
      I_Contact( "PUMP SELECTION"."P-301 RO 1 HPP PUMP B" )
      R_Coil( "MANUAL BIT"."P-301 B RO 1 HPP PUMP" )
   END_RUNG
   RUNG wire#powerrail
      Contact( "AlwaysTRUE" )
      wire#w3
      I_Contact( "PUMP SELECTION"."P-401 A RO 2 FEED PUMP" )
      R_Coil( "MANUAL BIT"."P-401 A RO 2 FEED PUMP" )
   END_RUNG
   RUNG wire#w3
      I_Contact( "PUMP SELECTION"."P-401 B RO 2 FEED PUMP" )
      R_Coil( "MANUAL BIT"."P-401 B RO 2 FEED PUMP" )
   END_RUNG
   RUNG wire#w3
      I_Contact( "PUMP SELECTION"."P-401 C RO 2 FEED PUMP" )
      R_Coil( "MANUAL BIT"."P-401 C RO 2 FEED PUMP" )
   END_RUNG
   RUNG wire#powerrail
      Contact( "AlwaysTRUE" )
      wire#w4
      I_Contact( "PUMP SELECTION"."P-402 RO 2 HPP A" )
      R_Coil( "MANUAL BIT"."P-402  A RO 2 HPP" )
   END_RUNG
   RUNG wire#w4
      I_Contact( "PUMP SELECTION"."P-402 RO 2 HPP B" )
      R_Coil( "MANUAL BIT"."P-402 B" )
   END_RUNG
   RUNG wire#powerrail
      Contact( "AlwaysTRUE" )
      wire#w5
      I_Contact( "PUMP SELECTION"."P-501 A EDI FEED PUMP" )
      R_Coil( "MANUAL BIT"."P-501 A EDI FEED PUMP" )
   END_RUNG
   RUNG wire#w5
      I_Contact( "PUMP SELECTION"."P-501 B EDI FEED PUMP" )
      R_Coil( "MANUAL BIT"."P-501 B EDI FEED PUMP" )
   END_RUNG
   RUNG wire#w5
      I_Contact( "PUMP SELECTION"."P-501 C EDI FEED PUMP" )
      R_Coil( "MANUAL BIT"."P-501 C EDI FEED PUMP" )
   END_RUNG
   RUNG wire#powerrail
      Contact( "AlwaysTRUE" )
      wire#w6
      I_Contact( "PUMP SELECTION"."EDI-501" )
      R_Coil( "MANUAL BIT"."EDI 501" )
   END_RUNG
   RUNG wire#w6
      I_Contact( "PUMP SELECTION"."EDI-502" )
      R_Coil( "MANUAL BIT"."EDI 502" )
   END_RUNG
   // the same network as SCL:
   IF "AlwaysTRUE" AND NOT "PUMP SELECTION"."P-202 A RO 1 FEED PUMP" THEN
       "MANUAL BIT"."P-202 A RO 1 FEED PUMP" := FALSE;
   END_IF;
   IF "AlwaysTRUE" AND NOT "PUMP SELECTION"."P-202 B RO 1 FEED PUMP" THEN
       "MANUAL BIT"."P-202 B RO 1 FEED PUMP" := FALSE;
   END_IF;
   IF "AlwaysTRUE" AND NOT "PUMP SELECTION"."P-202 C RO 1 FEED PUMP" THEN
       "MANUAL BIT"."P-202 C RO 1 FEED PUMP" := FALSE;
   END_IF;
   IF "AlwaysTRUE" AND NOT "PUMP SELECTION"."P-301 RO 1 HPP PUMP A" THEN
       "MANUAL BIT"."P-301 A RO 1 HPP PUMP" := FALSE;
   END_IF;
   IF "AlwaysTRUE" AND NOT "PUMP SELECTION"."P-301 RO 1 HPP PUMP B" THEN
       "MANUAL BIT"."P-301 B RO 1 HPP PUMP" := FALSE;
   END_IF;
   IF "AlwaysTRUE" AND NOT "PUMP SELECTION"."P-401 A RO 2 FEED PUMP" THEN
       "MANUAL BIT"."P-401 A RO 2 FEED PUMP" := FALSE;
   END_IF;
   IF "AlwaysTRUE" AND NOT "PUMP SELECTION"."P-401 B RO 2 FEED PUMP" THEN
       "MANUAL BIT"."P-401 B RO 2 FEED PUMP" := FALSE;
   END_IF;
   IF "AlwaysTRUE" AND NOT "PUMP SELECTION"."P-401 C RO 2 FEED PUMP" THEN
       "MANUAL BIT"."P-401 C RO 2 FEED PUMP" := FALSE;
   END_IF;
   IF "AlwaysTRUE" AND NOT "PUMP SELECTION"."P-402 RO 2 HPP A" THEN
       "MANUAL BIT"."P-402  A RO 2 HPP" := FALSE;
   END_IF;
   IF "AlwaysTRUE" AND NOT "PUMP SELECTION"."P-402 RO 2 HPP B" THEN "MANUAL BIT"."P-402 B" := FALSE; END_IF;
   IF "AlwaysTRUE" AND NOT "PUMP SELECTION"."P-501 A EDI FEED PUMP" THEN
       "MANUAL BIT"."P-501 A EDI FEED PUMP" := FALSE;
   END_IF;
   IF "AlwaysTRUE" AND NOT "PUMP SELECTION"."P-501 B EDI FEED PUMP" THEN
       "MANUAL BIT"."P-501 B EDI FEED PUMP" := FALSE;
   END_IF;
   IF "AlwaysTRUE" AND NOT "PUMP SELECTION"."P-501 C EDI FEED PUMP" THEN
       "MANUAL BIT"."P-501 C EDI FEED PUMP" := FALSE;
   END_IF;
   IF "AlwaysTRUE" AND NOT "PUMP SELECTION"."EDI-501" THEN "MANUAL BIT"."EDI 501" := FALSE; END_IF;
   IF "AlwaysTRUE" AND NOT "PUMP SELECTION"."EDI-502" THEN "MANUAL BIT"."EDI 502" := FALSE; END_IF;
END_REGION

REGION Network 10: AUTO INTERLOCK FOR RO-1 ///////////////////////////////////////////////////////
END_REGION

REGION Network 11: CEB1 AND CEB2 SYSTEM IN RUNNING AFTER RO SYSTEM HOLD
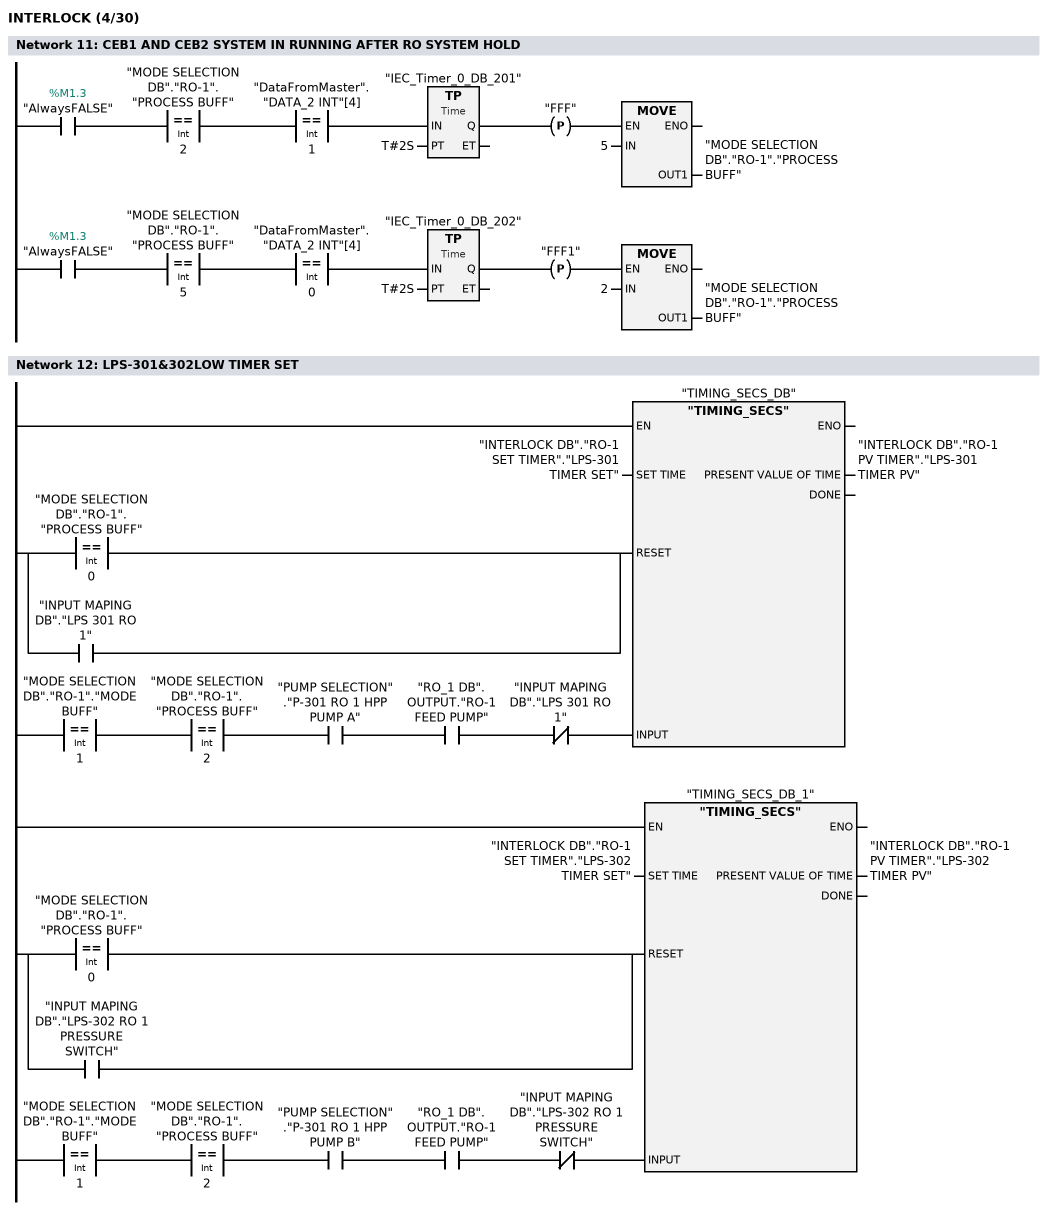
   RUNG wire#powerrail
      Contact( "AlwaysFALSE" )
      { S7_Templates := "SrcType := Int" } EQ_Contact(in1 := "MODE SELECTION DB"."RO-1"."PROCESS BUFF", in2 := 2)
      { S7_Templates := "SrcType := Int" } EQ_Contact(in1 := "DataFromMaster"."DATA_2 INT"[4], in2 := 1)
      { S7_Templates := "time_type := Time" } "IEC_Timer_0_DB_201".TP(pt := T#2S, et =>)
      P_Trig( "FFF" )
      Move(in := 5, out1 => "MODE SELECTION DB"."RO-1"."PROCESS BUFF")
   END_RUNG
   RUNG wire#powerrail
      Contact( "AlwaysFALSE" )
      { S7_Templates := "SrcType := Int" } EQ_Contact(in1 := "MODE SELECTION DB"."RO-1"."PROCESS BUFF", in2 := 5)
      { S7_Templates := "SrcType := Int" } EQ_Contact(in1 := "DataFromMaster"."DATA_2 INT"[4], in2 := 0)
      { S7_Templates := "time_type := Time" } "IEC_Timer_0_DB_202".TP(pt := T#2S, et =>)
      P_Trig( "FFF1" )
      Move(in := 2, out1 => "MODE SELECTION DB"."RO-1"."PROCESS BUFF")
   END_RUNG
   // the same network as SCL:
   "IEC_Timer_0_DB_201".TP(IN := "AlwaysFALSE" AND ("MODE SELECTION DB"."RO-1"."PROCESS BUFF" = 2) AND ("DataFromMaster"."DATA_2 INT"[4] = 1),
                           PT := T#2S);
   #_w1 := "IEC_Timer_0_DB_201".Q AND NOT "FFF";   // rising edge
   "FFF" := "IEC_Timer_0_DB_201".Q;
   IF #_w1 THEN "MODE SELECTION DB"."RO-1"."PROCESS BUFF" := 5; END_IF;
   "IEC_Timer_0_DB_202".TP(IN := "AlwaysFALSE" AND ("MODE SELECTION DB"."RO-1"."PROCESS BUFF" = 5) AND ("DataFromMaster"."DATA_2 INT"[4] = 0),
                           PT := T#2S);
   #_w2 := "IEC_Timer_0_DB_202".Q AND NOT "FFF1";   // rising edge
   "FFF1" := "IEC_Timer_0_DB_202".Q;
   IF #_w2 THEN "MODE SELECTION DB"."RO-1"."PROCESS BUFF" := 2; END_IF;
END_REGION

REGION Network 12: LPS-301&302LOW TIMER SET
   RUNG wire#powerrail
      "TIMING_SECS_DB"(RESET := wire#w1, INPUT := wire#w2, "SET TIME" := "INTERLOCK DB"."RO-1 SET TIMER"."LPS-301 TIMER SET", "PRESENT VALUE OF TIME" => "INTERLOCK DB"."RO-1 PV TIMER"."LPS-301 TIMER PV", DONE =>)
   END_RUNG
   RUNG wire#powerrail
      { S7_Templates := "SrcType := Int" } EQ_Contact(in1 := "MODE SELECTION DB"."RO-1"."PROCESS BUFF", in2 := 0)
   END_RUNG wire#w1
   RUNG wire#powerrail
      Contact( "INPUT MAPING DB"."LPS 301 RO 1" )
   END_RUNG wire#w1
   RUNG wire#powerrail
      { S7_Templates := "SrcType := Int" } EQ_Contact(in1 := "MODE SELECTION DB"."RO-1"."MODE BUFF", in2 := 1)
      { S7_Templates := "SrcType := Int" } EQ_Contact(in1 := "MODE SELECTION DB"."RO-1"."PROCESS BUFF", in2 := 2)
      Contact( "PUMP SELECTION"."P-301 RO 1 HPP PUMP A" )
      Contact( "RO_1 DB".OUTPUT."RO-1 FEED PUMP" )
      I_Contact( "INPUT MAPING DB"."LPS 301 RO 1" )
   END_RUNG wire#w2
   RUNG wire#powerrail
      "TIMING_SECS_DB_1"(RESET := wire#w3, INPUT := wire#w4, "SET TIME" := "INTERLOCK DB"."RO-1 SET TIMER"."LPS-302 TIMER SET", "PRESENT VALUE OF TIME" => "INTERLOCK DB"."RO-1 PV TIMER"."LPS-302 TIMER PV", DONE =>)
   END_RUNG
   RUNG wire#powerrail
      { S7_Templates := "SrcType := Int" } EQ_Contact(in1 := "MODE SELECTION DB"."RO-1"."PROCESS BUFF", in2 := 0)
   END_RUNG wire#w3
   RUNG wire#powerrail
      Contact( "INPUT MAPING DB"."LPS-302 RO 1 PRESSURE SWITCH" )
   END_RUNG wire#w3
   RUNG wire#powerrail
      { S7_Templates := "SrcType := Int" } EQ_Contact(in1 := "MODE SELECTION DB"."RO-1"."MODE BUFF", in2 := 1)
      { S7_Templates := "SrcType := Int" } EQ_Contact(in1 := "MODE SELECTION DB"."RO-1"."PROCESS BUFF", in2 := 2)
      Contact( "PUMP SELECTION"."P-301 RO 1 HPP PUMP B" )
      Contact( "RO_1 DB".OUTPUT."RO-1 FEED PUMP" )
      I_Contact( "INPUT MAPING DB"."LPS-302 RO 1 PRESSURE SWITCH" )
   END_RUNG wire#w4
   // the same network as SCL:
   "TIMING_SECS_DB"("SET TIME" := "INTERLOCK DB"."RO-1 SET TIMER"."LPS-301 TIMER SET",   // "TIMING_SECS"
                    RESET := ("MODE SELECTION DB"."RO-1"."PROCESS BUFF" = 0) OR "INPUT MAPING DB"."LPS 301 RO 1",
                    INPUT := ("MODE SELECTION DB"."RO-1"."MODE BUFF" = 1) AND ("MODE SELECTION DB"."RO-1"."PROCESS BUFF" = 2) AND "PUMP SELECTION"."P-301 RO 1 HPP PUMP A" AND "RO_1 DB".OUTPUT."RO-1 FEED PUMP" AND NOT "INPUT MAPING DB"."LPS 301 RO 1",
                    "PRESENT VALUE OF TIME" => "INTERLOCK DB"."RO-1 PV TIMER"."LPS-301 TIMER PV");
   "TIMING_SECS_DB_1"("SET TIME" := "INTERLOCK DB"."RO-1 SET TIMER"."LPS-302 TIMER SET",   // "TIMING_SECS"
                      RESET := ("MODE SELECTION DB"."RO-1"."PROCESS BUFF" = 0) OR "INPUT MAPING DB"."LPS-302 RO 1 PRESSURE SWITCH",
                      INPUT := ("MODE SELECTION DB"."RO-1"."MODE BUFF" = 1) AND ("MODE SELECTION DB"."RO-1"."PROCESS BUFF" = 2) AND "PUMP SELECTION"."P-301 RO 1 HPP PUMP B" AND "RO_1 DB".OUTPUT."RO-1 FEED PUMP" AND NOT "INPUT MAPING DB"."LPS-302 RO 1 PRESSURE SWITCH",
                      "PRESENT VALUE OF TIME" => "INTERLOCK DB"."RO-1 PV TIMER"."LPS-302 TIMER PV");
END_REGION

REGION Network 13: HPS-301 &302
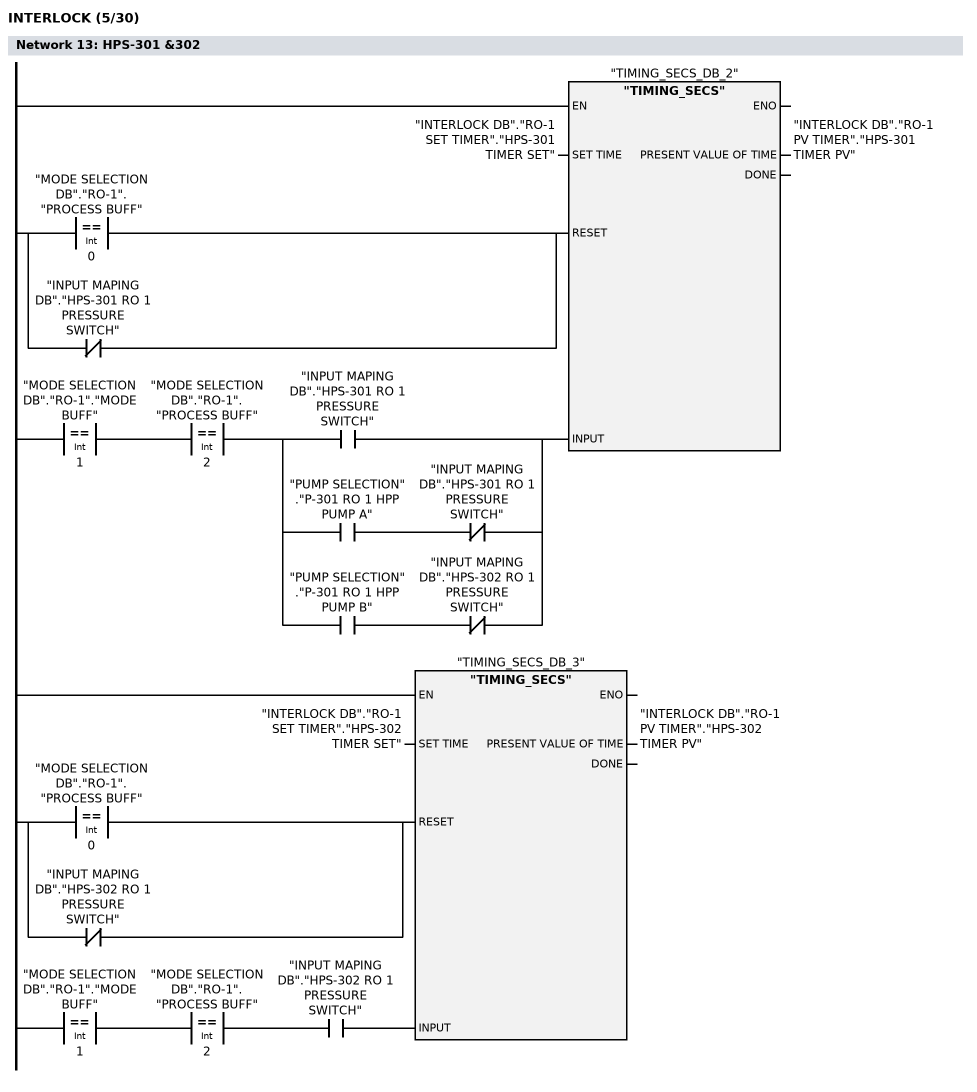
   RUNG wire#powerrail
      "TIMING_SECS_DB_2"(RESET := wire#w1, INPUT := wire#w3, "SET TIME" := "INTERLOCK DB"."RO-1 SET TIMER"."HPS-301 TIMER SET", "PRESENT VALUE OF TIME" => "INTERLOCK DB"."RO-1 PV TIMER"."HPS-301 TIMER PV", DONE =>)
   END_RUNG
   RUNG wire#powerrail
      { S7_Templates := "SrcType := Int" } EQ_Contact(in1 := "MODE SELECTION DB"."RO-1"."PROCESS BUFF", in2 := 0)
   END_RUNG wire#w1
   RUNG wire#powerrail
      I_Contact( "INPUT MAPING DB"."HPS-301 RO 1 PRESSURE SWITCH" )
   END_RUNG wire#w1
   RUNG wire#powerrail
      { S7_Templates := "SrcType := Int" } EQ_Contact(in1 := "MODE SELECTION DB"."RO-1"."MODE BUFF", in2 := 1)
      { S7_Templates := "SrcType := Int" } EQ_Contact(in1 := "MODE SELECTION DB"."RO-1"."PROCESS BUFF", in2 := 2)
      wire#w2
      Contact( "INPUT MAPING DB"."HPS-301 RO 1 PRESSURE SWITCH" )
   END_RUNG wire#w3
   RUNG wire#w2
      Contact( "PUMP SELECTION"."P-301 RO 1 HPP PUMP A" )
      I_Contact( "INPUT MAPING DB"."HPS-301 RO 1 PRESSURE SWITCH" )
   END_RUNG wire#w3
   RUNG wire#w2
      Contact( "PUMP SELECTION"."P-301 RO 1 HPP PUMP B" )
      I_Contact( "INPUT MAPING DB"."HPS-302 RO 1 PRESSURE SWITCH" )
   END_RUNG wire#w3
   RUNG wire#powerrail
      "TIMING_SECS_DB_3"(RESET := wire#w4, INPUT := wire#w5, "SET TIME" := "INTERLOCK DB"."RO-1 SET TIMER"."HPS-302 TIMER SET", "PRESENT VALUE OF TIME" => "INTERLOCK DB"."RO-1 PV TIMER"."HPS-302 TIMER PV", DONE =>)
   END_RUNG
   RUNG wire#powerrail
      { S7_Templates := "SrcType := Int" } EQ_Contact(in1 := "MODE SELECTION DB"."RO-1"."PROCESS BUFF", in2 := 0)
   END_RUNG wire#w4
   RUNG wire#powerrail
      I_Contact( "INPUT MAPING DB"."HPS-302 RO 1 PRESSURE SWITCH" )
   END_RUNG wire#w4
   RUNG wire#powerrail
      { S7_Templates := "SrcType := Int" } EQ_Contact(in1 := "MODE SELECTION DB"."RO-1"."MODE BUFF", in2 := 1)
      { S7_Templates := "SrcType := Int" } EQ_Contact(in1 := "MODE SELECTION DB"."RO-1"."PROCESS BUFF", in2 := 2)
      Contact( "INPUT MAPING DB"."HPS-302 RO 1 PRESSURE SWITCH" )
   END_RUNG wire#w5
   // the same network as SCL:
   "TIMING_SECS_DB_2"("SET TIME" := "INTERLOCK DB"."RO-1 SET TIMER"."HPS-301 TIMER SET",   // "TIMING_SECS"
                      RESET := ("MODE SELECTION DB"."RO-1"."PROCESS BUFF" = 0) OR NOT "INPUT MAPING DB"."HPS-301 RO 1 PRESSURE SWITCH",
                      INPUT := ("MODE SELECTION DB"."RO-1"."MODE BUFF" = 1) AND ("MODE SELECTION DB"."RO-1"."PROCESS BUFF" = 2) AND ("INPUT MAPING DB"."HPS-301 RO 1 PRESSURE SWITCH" OR ("PUMP SELECTION"."P-301 RO 1 HPP PUMP A" AND NOT "INPUT MAPING DB"."HPS-301 RO 1 PRESSURE SWITCH") OR ("PUMP SELECTION"."P-301 RO 1 HPP PUMP B" AND NOT "INPUT MAPING DB"."HPS-302 RO 1 PRESSURE SWITCH")),
                      "PRESENT VALUE OF TIME" => "INTERLOCK DB"."RO-1 PV TIMER"."HPS-301 TIMER PV");
   "TIMING_SECS_DB_3"("SET TIME" := "INTERLOCK DB"."RO-1 SET TIMER"."HPS-302 TIMER SET",   // "TIMING_SECS"
                      RESET := ("MODE SELECTION DB"."RO-1"."PROCESS BUFF" = 0) OR NOT "INPUT MAPING DB"."HPS-302 RO 1 PRESSURE SWITCH",
                      INPUT := ("MODE SELECTION DB"."RO-1"."MODE BUFF" = 1) AND ("MODE SELECTION DB"."RO-1"."PROCESS BUFF" = 2) AND "INPUT MAPING DB"."HPS-302 RO 1 PRESSURE SWITCH",
                      "PRESENT VALUE OF TIME" => "INTERLOCK DB"."RO-1 PV TIMER"."HPS-302 TIMER PV");
END_REGION

REGION Network 14: pH-301 HIGH/ LOW
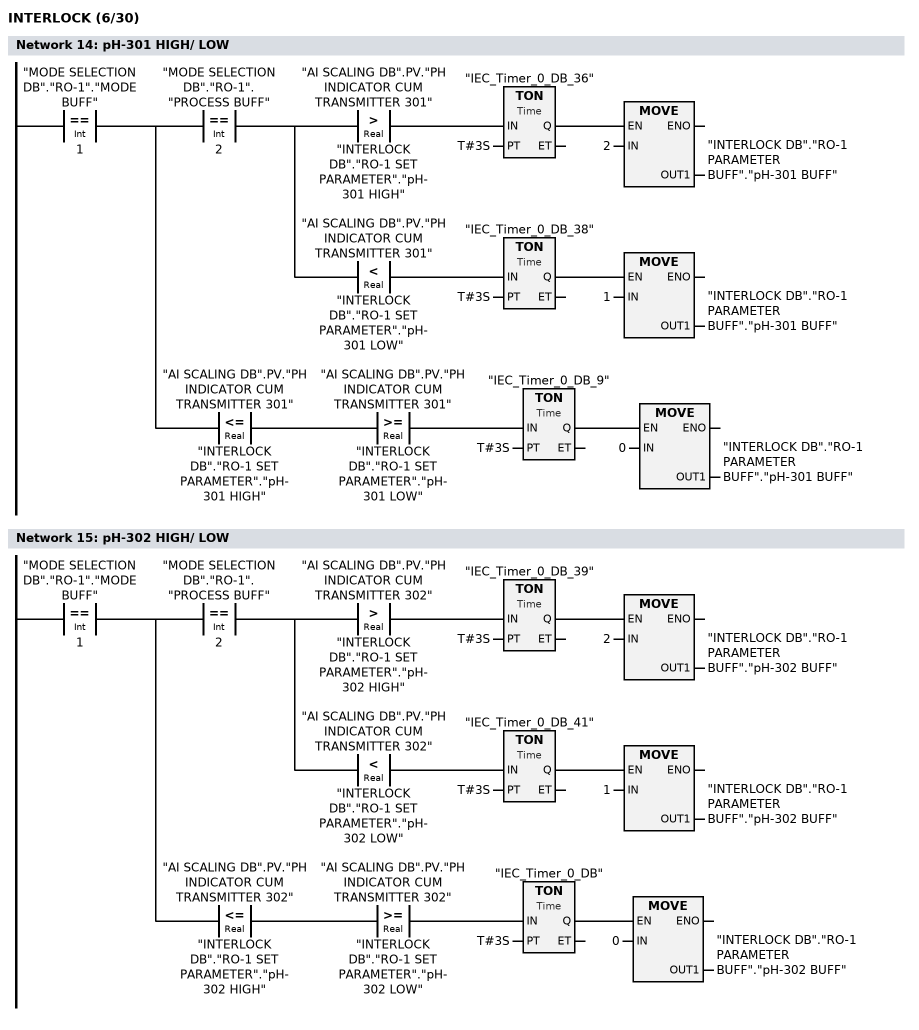
   RUNG wire#powerrail
      { S7_Templates := "SrcType := Int" } EQ_Contact(in1 := "MODE SELECTION DB"."RO-1"."MODE BUFF", in2 := 1)
      wire#w1
      { S7_Templates := "SrcType := Int" } EQ_Contact(in1 := "MODE SELECTION DB"."RO-1"."PROCESS BUFF", in2 := 2)
      wire#w2
      { S7_Templates := "SrcType := Real" } GT_Contact(in1 := "AI SCALING DB".PV."PH INDICATOR CUM TRANSMITTER 301", in2 := "INTERLOCK DB"."RO-1 SET PARAMETER"."pH-301 HIGH")
      { S7_Templates := "time_type := Time" } "IEC_Timer_0_DB_36".TON(pt := T#3S, et =>)
      Move(in := 2, out1 => "INTERLOCK DB"."RO-1 PARAMETER BUFF"."pH-301 BUFF")
   END_RUNG
   RUNG wire#w2
      { S7_Templates := "SrcType := Real" } LT_Contact(in1 := "AI SCALING DB".PV."PH INDICATOR CUM TRANSMITTER 301", in2 := "INTERLOCK DB"."RO-1 SET PARAMETER"."pH-301 LOW")
      { S7_Templates := "time_type := Time" } "IEC_Timer_0_DB_38".TON(pt := T#3S, et =>)
      Move(in := 1, out1 => "INTERLOCK DB"."RO-1 PARAMETER BUFF"."pH-301 BUFF")
   END_RUNG
   RUNG wire#w1
      { S7_Templates := "SrcType := Real" } LE_Contact(in1 := "AI SCALING DB".PV."PH INDICATOR CUM TRANSMITTER 301", in2 := "INTERLOCK DB"."RO-1 SET PARAMETER"."pH-301 HIGH")
      { S7_Templates := "SrcType := Real" } GE_Contact(in1 := "AI SCALING DB".PV."PH INDICATOR CUM TRANSMITTER 301", in2 := "INTERLOCK DB"."RO-1 SET PARAMETER"."pH-301 LOW")
      { S7_Templates := "time_type := Time" } "IEC_Timer_0_DB_9".TON(pt := T#3S, et =>)
      Move(in := 0, out1 => "INTERLOCK DB"."RO-1 PARAMETER BUFF"."pH-301 BUFF")
   END_RUNG
   // the same network as SCL:
   #_w1 := "MODE SELECTION DB"."RO-1"."MODE BUFF" = 1;
   #_w2 := #_w1 AND ("MODE SELECTION DB"."RO-1"."PROCESS BUFF" = 2);
   "IEC_Timer_0_DB_36".TON(IN := #_w2 AND ("AI SCALING DB".PV."PH INDICATOR CUM TRANSMITTER 301" > "INTERLOCK DB"."RO-1 SET PARAMETER"."pH-301 HIGH"),
                           PT := T#3S);
   IF "IEC_Timer_0_DB_36".Q THEN "INTERLOCK DB"."RO-1 PARAMETER BUFF"."pH-301 BUFF" := 2; END_IF;
   "IEC_Timer_0_DB_38".TON(IN := #_w2 AND ("AI SCALING DB".PV."PH INDICATOR CUM TRANSMITTER 301" < "INTERLOCK DB"."RO-1 SET PARAMETER"."pH-301 LOW"),
                           PT := T#3S);
   IF "IEC_Timer_0_DB_38".Q THEN "INTERLOCK DB"."RO-1 PARAMETER BUFF"."pH-301 BUFF" := 1; END_IF;
   "IEC_Timer_0_DB_9".TON(IN := #_w1 AND ("AI SCALING DB".PV."PH INDICATOR CUM TRANSMITTER 301" <= "INTERLOCK DB"."RO-1 SET PARAMETER"."pH-301 HIGH") AND ("AI SCALING DB".PV."PH INDICATOR CUM TRANSMITTER 301" >= "INTERLOCK DB"."RO-1 SET PARAMETER"."pH-301 LOW"),
                          PT := T#3S);
   IF "IEC_Timer_0_DB_9".Q THEN "INTERLOCK DB"."RO-1 PARAMETER BUFF"."pH-301 BUFF" := 0; END_IF;
END_REGION

REGION Network 15: pH-302 HIGH/ LOW
   RUNG wire#powerrail
      { S7_Templates := "SrcType := Int" } EQ_Contact(in1 := "MODE SELECTION DB"."RO-1"."MODE BUFF", in2 := 1)
      wire#w1
      { S7_Templates := "SrcType := Int" } EQ_Contact(in1 := "MODE SELECTION DB"."RO-1"."PROCESS BUFF", in2 := 2)
      wire#w2
      { S7_Templates := "SrcType := Real" } GT_Contact(in1 := "AI SCALING DB".PV."PH INDICATOR CUM TRANSMITTER 302", in2 := "INTERLOCK DB"."RO-1 SET PARAMETER"."pH-302 HIGH")
      { S7_Templates := "time_type := Time" } "IEC_Timer_0_DB_39".TON(pt := T#3S, et =>)
      Move(in := 2, out1 => "INTERLOCK DB"."RO-1 PARAMETER BUFF"."pH-302 BUFF")
   END_RUNG
   RUNG wire#w2
      { S7_Templates := "SrcType := Real" } LT_Contact(in1 := "AI SCALING DB".PV."PH INDICATOR CUM TRANSMITTER 302", in2 := "INTERLOCK DB"."RO-1 SET PARAMETER"."pH-302 LOW")
      { S7_Templates := "time_type := Time" } "IEC_Timer_0_DB_41".TON(pt := T#3S, et =>)
      Move(in := 1, out1 => "INTERLOCK DB"."RO-1 PARAMETER BUFF"."pH-302 BUFF")
   END_RUNG
   RUNG wire#w1
      { S7_Templates := "SrcType := Real" } LE_Contact(in1 := "AI SCALING DB".PV."PH INDICATOR CUM TRANSMITTER 302", in2 := "INTERLOCK DB"."RO-1 SET PARAMETER"."pH-302 HIGH")
      { S7_Templates := "SrcType := Real" } GE_Contact(in1 := "AI SCALING DB".PV."PH INDICATOR CUM TRANSMITTER 302", in2 := "INTERLOCK DB"."RO-1 SET PARAMETER"."pH-302 LOW")
      { S7_Templates := "time_type := Time" } "IEC_Timer_0_DB".TON(pt := T#3S, et =>)
      Move(in := 0, out1 => "INTERLOCK DB"."RO-1 PARAMETER BUFF"."pH-302 BUFF")
   END_RUNG
   // the same network as SCL:
   #_w1 := "MODE SELECTION DB"."RO-1"."MODE BUFF" = 1;
   #_w2 := #_w1 AND ("MODE SELECTION DB"."RO-1"."PROCESS BUFF" = 2);
   "IEC_Timer_0_DB_39".TON(IN := #_w2 AND ("AI SCALING DB".PV."PH INDICATOR CUM TRANSMITTER 302" > "INTERLOCK DB"."RO-1 SET PARAMETER"."pH-302 HIGH"),
                           PT := T#3S);
   IF "IEC_Timer_0_DB_39".Q THEN "INTERLOCK DB"."RO-1 PARAMETER BUFF"."pH-302 BUFF" := 2; END_IF;
   "IEC_Timer_0_DB_41".TON(IN := #_w2 AND ("AI SCALING DB".PV."PH INDICATOR CUM TRANSMITTER 302" < "INTERLOCK DB"."RO-1 SET PARAMETER"."pH-302 LOW"),
                           PT := T#3S);
   IF "IEC_Timer_0_DB_41".Q THEN "INTERLOCK DB"."RO-1 PARAMETER BUFF"."pH-302 BUFF" := 1; END_IF;
   "IEC_Timer_0_DB".TON(IN := #_w1 AND ("AI SCALING DB".PV."PH INDICATOR CUM TRANSMITTER 302" <= "INTERLOCK DB"."RO-1 SET PARAMETER"."pH-302 HIGH") AND ("AI SCALING DB".PV."PH INDICATOR CUM TRANSMITTER 302" >= "INTERLOCK DB"."RO-1 SET PARAMETER"."pH-302 LOW"),
                        PT := T#3S);
   IF "IEC_Timer_0_DB".Q THEN "INTERLOCK DB"."RO-1 PARAMETER BUFF"."pH-302 BUFF" := 0; END_IF;
END_REGION

REGION Network 16: CT-301 HIGH
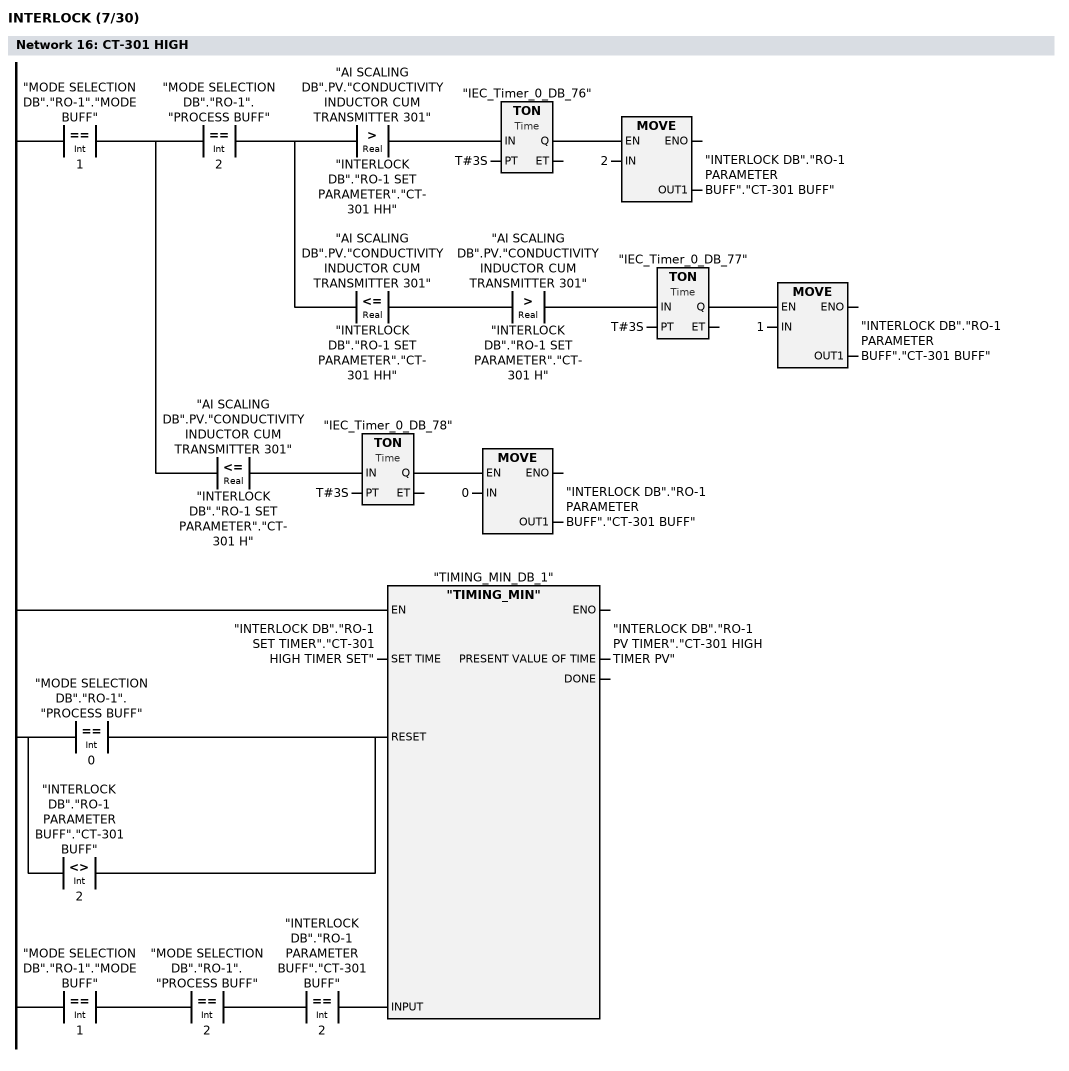
   RUNG wire#powerrail
      { S7_Templates := "SrcType := Int" } EQ_Contact(in1 := "MODE SELECTION DB"."RO-1"."MODE BUFF", in2 := 1)
      wire#w1
      { S7_Templates := "SrcType := Int" } EQ_Contact(in1 := "MODE SELECTION DB"."RO-1"."PROCESS BUFF", in2 := 2)
      wire#w2
      { S7_Templates := "SrcType := Real" } GT_Contact(in1 := "AI SCALING DB".PV."CONDUCTIVITY INDUCTOR CUM TRANSMITTER 301", in2 := "INTERLOCK DB"."RO-1 SET PARAMETER"."CT-301 HH")
      { S7_Templates := "time_type := Time" } "IEC_Timer_0_DB_76".TON(pt := T#3S, et =>)
      Move(in := 2, out1 => "INTERLOCK DB"."RO-1 PARAMETER BUFF"."CT-301 BUFF")
   END_RUNG
   RUNG wire#w2
      { S7_Templates := "SrcType := Real" } LE_Contact(in1 := "AI SCALING DB".PV."CONDUCTIVITY INDUCTOR CUM TRANSMITTER 301", in2 := "INTERLOCK DB"."RO-1 SET PARAMETER"."CT-301 HH")
      { S7_Templates := "SrcType := Real" } GT_Contact(in1 := "AI SCALING DB".PV."CONDUCTIVITY INDUCTOR CUM TRANSMITTER 301", in2 := "INTERLOCK DB"."RO-1 SET PARAMETER"."CT-301 H")
      { S7_Templates := "time_type := Time" } "IEC_Timer_0_DB_77".TON(pt := T#3S, et =>)
      Move(in := 1, out1 => "INTERLOCK DB"."RO-1 PARAMETER BUFF"."CT-301 BUFF")
   END_RUNG
   RUNG wire#w1
      { S7_Templates := "SrcType := Real" } LE_Contact(in1 := "AI SCALING DB".PV."CONDUCTIVITY INDUCTOR CUM TRANSMITTER 301", in2 := "INTERLOCK DB"."RO-1 SET PARAMETER"."CT-301 H")
      { S7_Templates := "time_type := Time" } "IEC_Timer_0_DB_78".TON(pt := T#3S, et =>)
      Move(in := 0, out1 => "INTERLOCK DB"."RO-1 PARAMETER BUFF"."CT-301 BUFF")
   END_RUNG
   RUNG wire#powerrail
      "TIMING_MIN_DB_1"(RESET := wire#w3, INPUT := wire#w4, "SET TIME" := "INTERLOCK DB"."RO-1 SET TIMER"."CT-301 HIGH TIMER SET", "PRESENT VALUE OF TIME" => "INTERLOCK DB"."RO-1 PV TIMER"."CT-301 HIGH TIMER PV", DONE =>)
   END_RUNG
   RUNG wire#powerrail
      { S7_Templates := "SrcType := Int" } EQ_Contact(in1 := "MODE SELECTION DB"."RO-1"."PROCESS BUFF", in2 := 0)
   END_RUNG wire#w3
   RUNG wire#powerrail
      { S7_Templates := "SrcType := Int" } NE_Contact(in1 := "INTERLOCK DB"."RO-1 PARAMETER BUFF"."CT-301 BUFF", in2 := 2)
   END_RUNG wire#w3
   RUNG wire#powerrail
      { S7_Templates := "SrcType := Int" } EQ_Contact(in1 := "MODE SELECTION DB"."RO-1"."MODE BUFF", in2 := 1)
      { S7_Templates := "SrcType := Int" } EQ_Contact(in1 := "MODE SELECTION DB"."RO-1"."PROCESS BUFF", in2 := 2)
      { S7_Templates := "SrcType := Int" } EQ_Contact(in1 := "INTERLOCK DB"."RO-1 PARAMETER BUFF"."CT-301 BUFF", in2 := 2)
   END_RUNG wire#w4
   // the same network as SCL:
   #_w1 := "MODE SELECTION DB"."RO-1"."MODE BUFF" = 1;
   #_w2 := #_w1 AND ("MODE SELECTION DB"."RO-1"."PROCESS BUFF" = 2);
   "IEC_Timer_0_DB_76".TON(IN := #_w2 AND ("AI SCALING DB".PV."CONDUCTIVITY INDUCTOR CUM TRANSMITTER 301" > "INTERLOCK DB"."RO-1 SET PARAMETER"."CT-301 HH"),
                           PT := T#3S);
   IF "IEC_Timer_0_DB_76".Q THEN "INTERLOCK DB"."RO-1 PARAMETER BUFF"."CT-301 BUFF" := 2; END_IF;
   "IEC_Timer_0_DB_77".TON(IN := #_w2 AND ("AI SCALING DB".PV."CONDUCTIVITY INDUCTOR CUM TRANSMITTER 301" <= "INTERLOCK DB"."RO-1 SET PARAMETER"."CT-301 HH") AND ("AI SCALING DB".PV."CONDUCTIVITY INDUCTOR CUM TRANSMITTER 301" > "INTERLOCK DB"."RO-1 SET PARAMETER"."CT-301 H"),
                           PT := T#3S);
   IF "IEC_Timer_0_DB_77".Q THEN "INTERLOCK DB"."RO-1 PARAMETER BUFF"."CT-301 BUFF" := 1; END_IF;
   "IEC_Timer_0_DB_78".TON(IN := #_w1 AND ("AI SCALING DB".PV."CONDUCTIVITY INDUCTOR CUM TRANSMITTER 301" <= "INTERLOCK DB"."RO-1 SET PARAMETER"."CT-301 H"),
                           PT := T#3S);
   IF "IEC_Timer_0_DB_78".Q THEN "INTERLOCK DB"."RO-1 PARAMETER BUFF"."CT-301 BUFF" := 0; END_IF;
   "TIMING_MIN_DB_1"("SET TIME" := "INTERLOCK DB"."RO-1 SET TIMER"."CT-301 HIGH TIMER SET",   // "TIMING_MIN"
                     RESET := ("MODE SELECTION DB"."RO-1"."PROCESS BUFF" = 0) OR ("INTERLOCK DB"."RO-1 PARAMETER BUFF"."CT-301 BUFF" <> 2),
                     INPUT := ("MODE SELECTION DB"."RO-1"."MODE BUFF" = 1) AND ("MODE SELECTION DB"."RO-1"."PROCESS BUFF" = 2) AND ("INTERLOCK DB"."RO-1 PARAMETER BUFF"."CT-301 BUFF" = 2),
                     "PRESENT VALUE OF TIME" => "INTERLOCK DB"."RO-1 PV TIMER"."CT-301 HIGH TIMER PV");
END_REGION

REGION Network 17: CT-302 HIGH
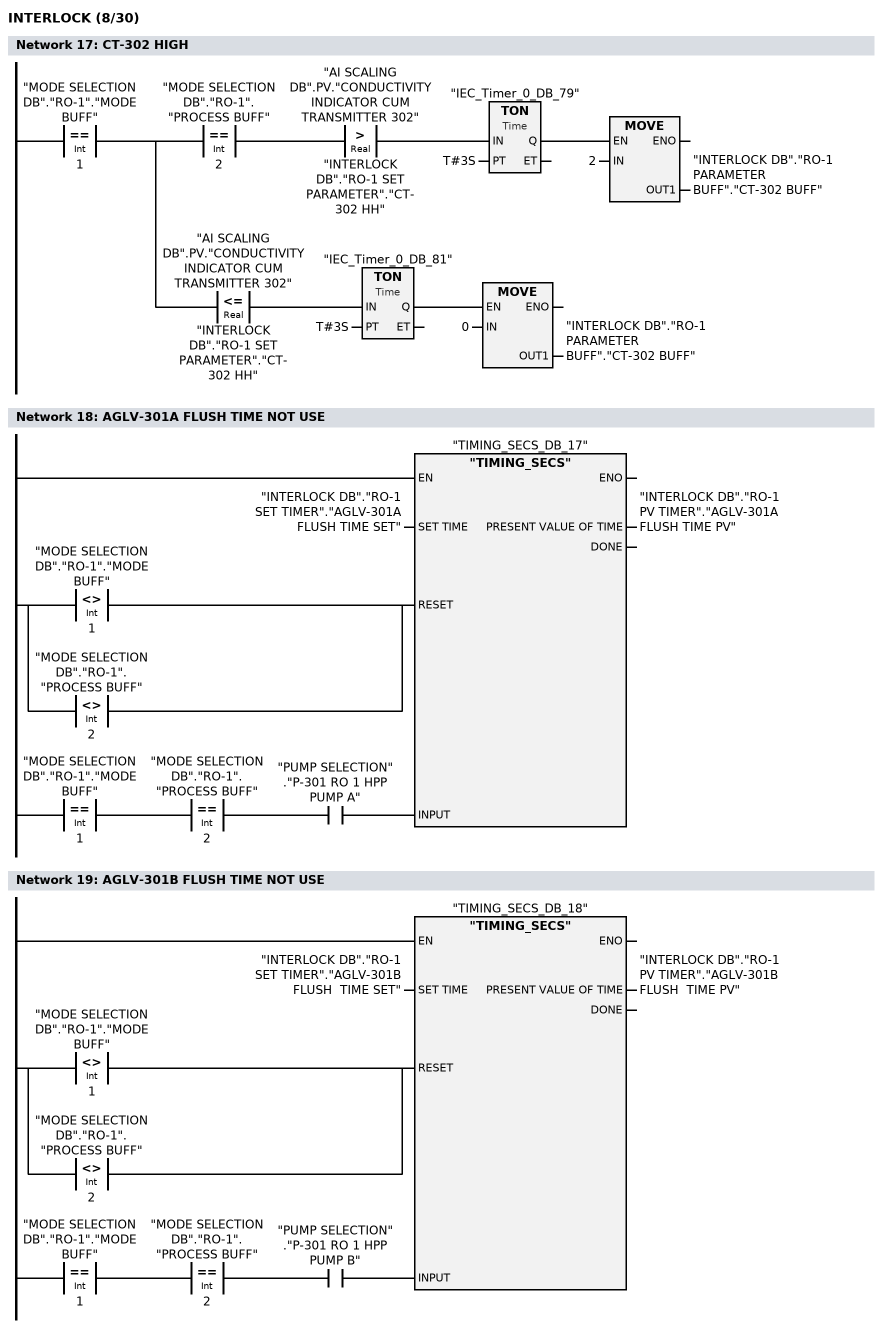
   RUNG wire#powerrail
      { S7_Templates := "SrcType := Int" } EQ_Contact(in1 := "MODE SELECTION DB"."RO-1"."MODE BUFF", in2 := 1)
      wire#w1
      { S7_Templates := "SrcType := Int" } EQ_Contact(in1 := "MODE SELECTION DB"."RO-1"."PROCESS BUFF", in2 := 2)
      { S7_Templates := "SrcType := Real" } GT_Contact(in1 := "AI SCALING DB".PV."CONDUCTIVITY INDICATOR CUM TRANSMITTER 302", in2 := "INTERLOCK DB"."RO-1 SET PARAMETER"."CT-302 HH")
      { S7_Templates := "time_type := Time" } "IEC_Timer_0_DB_79".TON(pt := T#3S, et =>)
      Move(in := 2, out1 => "INTERLOCK DB"."RO-1 PARAMETER BUFF"."CT-302 BUFF")
   END_RUNG
   RUNG wire#w1
      { S7_Templates := "SrcType := Real" } LE_Contact(in1 := "AI SCALING DB".PV."CONDUCTIVITY INDICATOR CUM TRANSMITTER 302", in2 := "INTERLOCK DB"."RO-1 SET PARAMETER"."CT-302 HH")
      { S7_Templates := "time_type := Time" } "IEC_Timer_0_DB_81".TON(pt := T#3S, et =>)
      Move(in := 0, out1 => "INTERLOCK DB"."RO-1 PARAMETER BUFF"."CT-302 BUFF")
   END_RUNG
   // the same network as SCL:
   #_w1 := "MODE SELECTION DB"."RO-1"."MODE BUFF" = 1;
   "IEC_Timer_0_DB_79".TON(IN := #_w1 AND ("MODE SELECTION DB"."RO-1"."PROCESS BUFF" = 2) AND ("AI SCALING DB".PV."CONDUCTIVITY INDICATOR CUM TRANSMITTER 302" > "INTERLOCK DB"."RO-1 SET PARAMETER"."CT-302 HH"),
                           PT := T#3S);
   IF "IEC_Timer_0_DB_79".Q THEN "INTERLOCK DB"."RO-1 PARAMETER BUFF"."CT-302 BUFF" := 2; END_IF;
   "IEC_Timer_0_DB_81".TON(IN := #_w1 AND ("AI SCALING DB".PV."CONDUCTIVITY INDICATOR CUM TRANSMITTER 302" <= "INTERLOCK DB"."RO-1 SET PARAMETER"."CT-302 HH"),
                           PT := T#3S);
   IF "IEC_Timer_0_DB_81".Q THEN "INTERLOCK DB"."RO-1 PARAMETER BUFF"."CT-302 BUFF" := 0; END_IF;
END_REGION

REGION Network 18: AGLV-301A FLUSH TIME NOT USE
   RUNG wire#powerrail
      "TIMING_SECS_DB_17"(RESET := wire#w1, INPUT := wire#w2, "SET TIME" := "INTERLOCK DB"."RO-1 SET TIMER"."AGLV-301A FLUSH TIME SET", "PRESENT VALUE OF TIME" => "INTERLOCK DB"."RO-1 PV TIMER"."AGLV-301A FLUSH TIME PV", DONE =>)
   END_RUNG
   RUNG wire#powerrail
      { S7_Templates := "SrcType := Int" } NE_Contact(in1 := "MODE SELECTION DB"."RO-1"."MODE BUFF", in2 := 1)
   END_RUNG wire#w1
   RUNG wire#powerrail
      { S7_Templates := "SrcType := Int" } NE_Contact(in1 := "MODE SELECTION DB"."RO-1"."PROCESS BUFF", in2 := 2)
   END_RUNG wire#w1
   RUNG wire#powerrail
      { S7_Templates := "SrcType := Int" } EQ_Contact(in1 := "MODE SELECTION DB"."RO-1"."MODE BUFF", in2 := 1)
      { S7_Templates := "SrcType := Int" } EQ_Contact(in1 := "MODE SELECTION DB"."RO-1"."PROCESS BUFF", in2 := 2)
      Contact( "PUMP SELECTION"."P-301 RO 1 HPP PUMP A" )
   END_RUNG wire#w2
   // the same network as SCL:
   "TIMING_SECS_DB_17"("SET TIME" := "INTERLOCK DB"."RO-1 SET TIMER"."AGLV-301A FLUSH TIME SET",   // "TIMING_SECS"
                       RESET := ("MODE SELECTION DB"."RO-1"."MODE BUFF" <> 1) OR ("MODE SELECTION DB"."RO-1"."PROCESS BUFF" <> 2),
                       INPUT := ("MODE SELECTION DB"."RO-1"."MODE BUFF" = 1) AND ("MODE SELECTION DB"."RO-1"."PROCESS BUFF" = 2) AND "PUMP SELECTION"."P-301 RO 1 HPP PUMP A",
                       "PRESENT VALUE OF TIME" => "INTERLOCK DB"."RO-1 PV TIMER"."AGLV-301A FLUSH TIME PV");
END_REGION

REGION Network 19: AGLV-301B FLUSH TIME NOT USE
   RUNG wire#powerrail
      "TIMING_SECS_DB_18"(RESET := wire#w1, INPUT := wire#w2, "SET TIME" := "INTERLOCK DB"."RO-1 SET TIMER"."AGLV-301B FLUSH  TIME SET", "PRESENT VALUE OF TIME" => "INTERLOCK DB"."RO-1 PV TIMER"."AGLV-301B FLUSH  TIME PV", DONE =>)
   END_RUNG
   RUNG wire#powerrail
      { S7_Templates := "SrcType := Int" } NE_Contact(in1 := "MODE SELECTION DB"."RO-1"."MODE BUFF", in2 := 1)
   END_RUNG wire#w1
   RUNG wire#powerrail
      { S7_Templates := "SrcType := Int" } NE_Contact(in1 := "MODE SELECTION DB"."RO-1"."PROCESS BUFF", in2 := 2)
   END_RUNG wire#w1
   RUNG wire#powerrail
      { S7_Templates := "SrcType := Int" } EQ_Contact(in1 := "MODE SELECTION DB"."RO-1"."MODE BUFF", in2 := 1)
      { S7_Templates := "SrcType := Int" } EQ_Contact(in1 := "MODE SELECTION DB"."RO-1"."PROCESS BUFF", in2 := 2)
      Contact( "PUMP SELECTION"."P-301 RO 1 HPP PUMP B" )
   END_RUNG wire#w2
   // the same network as SCL:
   "TIMING_SECS_DB_18"("SET TIME" := "INTERLOCK DB"."RO-1 SET TIMER"."AGLV-301B FLUSH  TIME SET",   // "TIMING_SECS"
                       RESET := ("MODE SELECTION DB"."RO-1"."MODE BUFF" <> 1) OR ("MODE SELECTION DB"."RO-1"."PROCESS BUFF" <> 2),
                       INPUT := ("MODE SELECTION DB"."RO-1"."MODE BUFF" = 1) AND ("MODE SELECTION DB"."RO-1"."PROCESS BUFF" = 2) AND "PUMP SELECTION"."P-301 RO 1 HPP PUMP B",
                       "PRESENT VALUE OF TIME" => "INTERLOCK DB"."RO-1 PV TIMER"."AGLV-301B FLUSH  TIME PV");
END_REGION

REGION Network 20: ORT-301
